# B&R Automation Studio project DeltaTestowa1 (part 2)

#### MainInitAction.st
```iecst
ACTION MainInitAction:

	MpPackMLCore_0.Enable := TRUE;
	MpPackMLMode_0.Enable := TRUE;
	MpDelta4Axis_0.Override := 100.0;
	MpDelta4Axis_0.Enable := TRUE;
	AxisParameters_0.Velocity := 50.0;
	AxisParameters_0.Acceleration := 20.0;
	AxisParameters_0.Deceleration := 20.0;

	AxisParameters_1.Velocity := 0.0;
	AxisParameters_1.Acceleration := 1.0;
	AxisParameters_1.Deceleration := 1.0;
	MpAxisBasic_0.Enable := TRUE;
	MpAxisBasic_1.Enable := TRUE;
	MpAxisBasic_Q1.Enable := TRUE;
	MpAxisBasic_Q2.Enable := TRUE;
	MpAxisBasic_Q3.Enable := TRUE;
	MpAxisBasic_Q4.Enable := TRUE;

	// dummy call of axis PVs just to avoid warning -2141192189 "The PV 'gAxisQx' does not exists" in logger
	gAxisQ1;
	gAxisQ2;
	gAxisQ3;
	gAxisQ4;

	IF DiagCpuIsARsim() THEN
		homingModeQ1.Homing.Mode := mcHOMING_DIRECT;
		homingModeQ2.Homing.Mode := mcHOMING_DIRECT;
		homingModeQ3.Homing.Mode := mcHOMING_DIRECT;
		homingModeQ4.Homing.Mode := mcHOMING_DIRECT;
	ELSE
		homingModeQ1.Homing.Mode := mcHOMING_DEFAULT;
		homingModeQ2.Homing.Mode := mcHOMING_DEFAULT;
		homingModeQ3.Homing.Mode := mcHOMING_DEFAULT;
		homingModeQ4.Homing.Mode := mcHOMING_DEFAULT;
	END_IF;

	//Activate block and set first state to Stopping (important, )
	MpPackMLMode_0.Activate := TRUE;
	MpPackMLMode_0.Stop := TRUE;

END_ACTION
```

#### MpPackCyclicAction.st
```iecst
ACTION MpPackCyclicAction:
	MpPackMLCore_0.MpLink := ADR(gPackMLCore);
	MpPackMLMode_0.MpLink := ADR(gPackMLCore);
	MpPackMLMode_0.ModeID := 1;

	MpPackMLMode_0.StateComplete := FALSE;
END_ACTION
```

#### AbortingAction.st
```iecst
ACTION AbortingAction:
	MpDelta4Axis_0.Power := FALSE;
	MpAxisBasic_0.Power := FALSE;
	ReadyMechanics := FALSE;
	AbortExecute := TRUE;
	CmdStart := FALSE;
	IF NOT MpDelta4Axis_0.PowerOn
		AND NOT MpAxisBasic_0.PowerOn THEN
		MpPackMLStateComplete(gPackMLCore,1);
	END_IF
END_ACTION
```

#### Action.st - not listed in the package file held
```iecst
ACTION ActionReseting:

	CASE RES_Step OF
		HOMING_DELTA:
			MpDelta4Axis_0.Home := TRUE;
			IF MpDelta4Axis_0.IsHomed THEN
				MpDelta4Axis_0.Home := FALSE;
				RES_Step := ACTIVATE_AXIS;
			END_IF

		ACTIVATE_AXIS:
			IF MpAxisBasic_0.Active AND MpDelta4Axis_0.Active THEN
				MpDelta4Axis_0.Power := TRUE;
				MpAxisBasic_0.Power := TRUE;
				MpAxisBasic_1.Power := TRUE; // axis not used, do not worry
				IF MpAxisBasic_0.PowerOn AND MpDelta4Axis_0.PowerOn THEN
					RES_Step := HOMING_AXIS;
				END_IF

			END_IF

		HOMING_AXIS:
			IF MpAxisBasic_0.PowerOn THEN
				MpAxisBasic_0.Home := TRUE;
				MpAxisBasic_1.Home := TRUE; // axis not used, do not worry
			END_IF;
			IF MpAxisBasic_0.IsHomed THEN
				MpAxisBasic_0.Home := FALSE;
				MpAxisBasic_1.Home := FALSE; // axis not used, do not worry
				RES_Step := COMPLETE_STATE;
			END_IF
		COMPLETE_STATE:
			MpPackMLStateComplete(gPackMLCore,1);

		END_CASE;
END_ACTION
```

### Program Logical/PickAndPlace/PrgPlace (IEC) - Place the products

#### Variables.var
```iecst
VAR
	P_Step : PlaceStepEnum;
	LastStep : PlaceStepEnum;
	Error : BOOL;
	PlaceHoldersSpacing : LREAL;
	LastPlaceHolderConveyorPosition : LREAL;
	ContainerID : UDINT;
	ElapsedDistance : LREAL;
END_VAR
(**)
(*Functionblocks*)
VAR
	MpPickRegister_0 : MpPickRegister;
	MpPickRegCreateContainer : MpPickRegCreateObject;
	MpPickRegGetObjectsContainer : MpPickRegGetObjects;
	MpPickRegDeleteTokens : MpPickRegDeleteObjects;
	Iterator : USINT;
	numberOfDeletes : USINT;
	TON_1 : TON;
	TON_0 : TON;
	OldTokenNumber : UDINT;
END_VAR
```

#### Main.st
```iecst
PROGRAM _INIT

    P_Step := P_WAIT_ENABLE;
    Error := FALSE;

	PlaceHoldersSpacing := 120; // distance between two consecutive place holders
	//numberOfDeletes := 2;
	gTokenNumber := 0;

END_PROGRAM

PROGRAM _CYCLIC

	IF NOT(gManualMode) THEN

	TON_0();
	TON_0.PT := T#5s;

    CASE P_Step OF
		P_WAIT_ENABLE:
			IF NOT AbortExecute AND NOT StopExecute AND NOT MpPickRegister_0.Error THEN
				P_Step := P_ENABLE_REGISTER_FB;
				StopExecutedPlace := FALSE;
				ClearingExecutedPlace := FALSE;
				MpPickRegister_0.ErrorReset := FALSE;
			END_IF

        P_ENABLE_REGISTER_FB:
            MpPickRegister_0.Enable := TRUE;
            P_Step := P_WAIT_ENABLE_REGISTER_FB;

        P_WAIT_ENABLE_REGISTER_FB:
            IF MpPickRegister_0.Active THEN
                P_Step := P_ENABLE_REGISTER_COMP;

            ELSIF MpPickRegister_0.Error THEN
                LastStep := P_Step;
                P_Step := P_ERROR;
            END_IF;

        P_ENABLE_REGISTER_COMP:
            MpPickRegister_0.RegisterEnable := TRUE;
            P_Step := P_WAIT_ENABLE_REGISTER_COMP;

        P_WAIT_ENABLE_REGISTER_COMP:
            IF MpPickRegister_0.RegisterActive THEN
                P_Step := P_ENABLE_ADD_REGISTER_FBS;

            ELSIF MpPickRegister_0.Error THEN
                LastStep := P_Step;
                P_Step := P_ERROR;
            END_IF;

        P_ENABLE_ADD_REGISTER_FBS:
            MpPickRegCreateContainer.Enable := TRUE;
			MpPickRegCreateContainer.Create := FALSE;
			MpPickRegGetObjectsContainer.Enable := TRUE;
			MpPickRegDeleteTokens.Enable := TRUE;
			P_Step := P_WAIT_ENABLE_ADD_REGISTER_FBS;

        P_WAIT_ENABLE_ADD_REGISTER_FBS:
            IF 	MpPickRegCreateContainer.Active THEN
                P_Step := P_WAIT_START_PROCESS;

            ELSIF MpPickRegCreateContainer.Error THEN
                LastStep := P_Step;
                P_Step := P_ERROR;
            END_IF;

        P_WAIT_START_PROCESS: // waits user start command and conveyor moving
            ReadyPlaceReg := TRUE;
            IF CmdStart AND ReadyToStart THEN
                P_Step := P_CREATE_OBJECTS;
            END_IF;

        (* We need to create positions (place holders) on place conveyor where to place picked objects *)
        P_CREATE_OBJECTS:

            ElapsedDistance := DistanceOverPeriod(PlaceConveyorPosition, LastPlaceHolderConveyorPosition, PlaceConveyorLength);

            IF (ElapsedDistance >= PlaceHoldersSpacing) THEN

                MpPickRegCreateContainer.Parameters.LatchedConveyor.Position := PlaceConveyorPosition;
                MpPickRegCreateContainer.Parameters.Mode := mpPICK_CREATE_CONTAINER_EMPTY;
				MpPickRegCreateContainer.Parameters.ObjectTypeName := 'MyContainer';
                MpPickRegCreateContainer.Parameters.Translation.X := 43;
				MpPickRegCreateContainer.Parameters.Translation.Y := 0;// in the middle of conveyor width
				MpPickRegCreateContainer.Parameters.Translation.Z := 2;
				ContainerID := MpPickRegCreateContainer.ObjectPositionId;
				MpPickRegCreateContainer.Create := TRUE;

				LastPlaceHolderConveyorPosition := MpPickRegCreateContainer.Parameters.LatchedConveyor.Position;
			ELSE
// Moze to trzeba rozwazyc ->ContainerID := MpPickRegCreateContainer.ObjectPositionId;
                MpPickRegCreateContainer.Create := FALSE;
            END_IF

        P_ERROR:
            Error := TRUE;
            ReadyPlaceReg := FALSE;

	END_CASE;

	IF StopExecute OR AbortExecute THEN
		ReadyPlaceReg := FALSE;
		P_Step := P_WAIT_ENABLE;
		StopExecutedPlace := TRUE;
	END_IF
	IF ClearingExecute THEN
		MpPickRegister_0.ErrorReset := TRUE;
		ClearingExecutedPlace := TRUE;
	END_IF

	MpPickRegGetObjectsContainer.Get := FALSE;
	MpPickRegDeleteTokens.Delete := FALSE;
	IF (MpPickRegGetObjectsContainer.Get = FALSE) THEN
		TON_0.IN := TRUE;

		IF TON_0.Q THEN
			MpPickRegGetObjectsContainer.Get := TRUE;
			TON_0.IN := FALSE;
		END_IF
	END_IF

	IF ContainerID > 0 THEN

		MpPickRegGetObjectsContainer.Parameters.DataAddress := ADR(gContainerInfo);
		MpPickRegGetObjectsContainer.Parameters.GetMode := mpPICK_GET_CONTAINER_CONTENT;
		MpPickRegGetObjectsContainer.Parameters.ObjectPositionId := ContainerID;
		MpPickRegGetObjectsContainer.Parameters.ObjectTypeName := 'MyContainer';
		MpPickRegGetObjectsContainer.Parameters.NumberOfObjectPositions := 4;
		MpPickRegGetObjectsContainer.MpLink := ADR(gPlaceRegister);
		MpPickRegGetObjectsContainer();

	END_IF;

		MpPickRegDeleteTokens.MpLink := ADR(gPlaceRegister);
		gTokenNumber := 0;

		FOR Iterator := 0 TO 3 DO
			IF (gContainerInfo[Iterator].ObjectPositionInfo = mpPICK_INFO_CONTAINED_OBJECT AND gDeleteObjects) THEN
				MpPickRegDeleteTokens.Parameters.ObjectTypeName := 'MyContainer';
				MpPickRegDeleteTokens.Parameters.ObjectPositionId := gContainerInfo[Iterator].ObjectPositionId;
				MpPickRegDeleteTokens.Delete := TRUE;
				numberOfDeletes := numberOfDeletes + 1;
			ELSE
				MpPickRegDeleteTokens.Parameters.ObjectTypeName := 'MyContainer';
				MpPickRegDeleteTokens.Parameters.ObjectPositionId := gContainerInfo[Iterator].ObjectPositionId;
				MpPickRegDeleteTokens.Delete := FALSE;
			END_IF;

			MpPickRegDeleteTokens();

			IF (gContainerInfo[Iterator].ObjectPositionInfo = mpPICK_INFO_CONTAINED_OBJECT) THEN
				gTokenNumber := gTokenNumber +1;
				IF OldTokenNumber <> gTokenNumber THEN
					gTokenOnConv := FALSE;
				END_IF

			END_IF

		END_FOR;
		IF numberOfDeletes > 0 THEN
			P_Step := P_WAIT_ENABLE;
			gTokenNumber := 0;
			numberOfDeletes := 0;
		END_IF
		gDeleteObjects := 0;
		OldTokenNumber := gTokenNumber;

		(* FB calls *)
		MpPickRegister_0.MpLink := ADR(gPlaceRegister);
		MpPickRegister_0();

		MpPickRegCreateContainer.MpLink := ADR(gPlaceRegister);
		MpPickRegCreateContainer();

	END_IF

END_PROGRAM
```

### Program Logical/PickAndPlace/PrgManual (IEC)

#### Types.typ
```iecst
TYPE
	MANUAL_ENUM :
		(
		HOMING := 1,
		XPOS := 2,
		XNEG := 3,
		YPOS := 4,
		YNEG := 5,
		ZPOS := 6,
		ZNEG := 7,
		OTHER := 8
		);
END_TYPE
```

#### Variables.var
```iecst
VAR
	HomeX : USINT;
	HomeY : USINT;
	HomingOffset : USINT;
	HomingVel : USINT;
	HomeZ : USINT;
	MoveXPos : BOOL;
	MoveXNeg : BOOL;
	MoveYPos : BOOL;
	MoveYNeg : BOOL;
	MoveZPos : BOOL;
	MoveZNeg : BOOL;
	XVel : USINT;
	YVel : USINT;
	ZVel : USINT;
	isMove : BOOL;
	ManualEnum : MANUAL_ENUM;
END_VAR
```

#### Main.st
```iecst
PROGRAM _INIT
	(* Insert code here *)
	gManualMode := 0;
	gMpDelta4AxisJog := FALSE;
	HomeX := 0;
	HomeY := 0;
	HomeZ := 120;
	HomingVel := 10;
	HomingOffset := 2;

END_PROGRAM

PROGRAM _CYCLIC
	IF gManualMode THEN
			//zapisac jako akcje:
		DeltaParamConnections.Jog.Velocity[0] := 0;
		DeltaParamConnections.Jog.Velocity[1] := 0;
		DeltaParamConnections.Jog.Velocity[2] := 0;

		IF isMove THEN
			gManualHoming := FALSE;
		END_IF;

		IF NOT isMove AND NOT gManualHoming THEN
			ManualEnum := 8;
		END_IF;

		IF gManualHoming THEN
			ManualEnum := 1;
		END_IF;

		gMpDelta4AxisEnable := TRUE;
		gMpDelta4AxisJog := TRUE;
		DeltaParamConnections.ManualMoveType := mcMOVE_RELATIVE;
		DeltaParamConnections.Jog.CoordSystem := mcTCS;
		DeltaParamConnections.CoordSystem := mcTCS;

		CASE ManualEnum OF
			HOMING:
				gMpDelta4AxisJog := TRUE;
				IF gTcpPositionX - HomeX > HomingOffset THEN
					DeltaParamConnections.Jog.Velocity[0] := -HomingVel;
				ELSIF HomeX - gTcpPositionX > HomingOffset THEN
					DeltaParamConnections.Jog.Velocity[0] := HomingVel;
				ELSIF gTcpPositionY - HomeY  > HomingOffset THEN
					DeltaParamConnections.Jog.Velocity[0] := 0;
					DeltaParamConnections.Jog.Velocity[1] := -HomingVel;
				ELSIF HomeY - gTcpPositionY > HomingOffset THEN
					DeltaParamConnections.Jog.Velocity[1] := HomingVel;
				ELSIF gTcpPositionZ - HomeZ > HomingOffset THEN
					DeltaParamConnections.Jog.Velocity[1] := 0;
					DeltaParamConnections.Jog.Velocity[2] := -HomingVel;
				ELSIF HomeZ - gTcpPositionZ > HomingOffset THEN
					DeltaParamConnections.Jog.Velocity[2] := HomingVel;
				ELSE
					DeltaParamConnections.Jog.Velocity[0] := 0;
					DeltaParamConnections.Jog.Velocity[1] := 0;
					DeltaParamConnections.Jog.Velocity[2] := 0;
				END_IF

			XPOS: DeltaParamConnections.Jog.Velocity[0] := XVel;
			XNEG: DeltaParamConnections.Jog.Velocity[0] := -XVel;
			YPOS: DeltaParamConnections.Jog.Velocity[1] := YVel;
			YNEG: DeltaParamConnections.Jog.Velocity[1] := -YVel;
			ZPOS: DeltaParamConnections.Jog.Velocity[2] := ZVel;
			ZNEG: DeltaParamConnections.Jog.Velocity[2] := -ZVel;
			OTHER: gMpDelta4AxisJog := FALSE;
			END_CASE

END_IF

END_PROGRAM
```

### Program Logical/PickAndPlace/Audyt (IEC)

#### Variables.var
```iecst
VAR
	MpAuditTrail_0 : MpAuditTrail;
	TypeVar : WSTRING[100];
	MessageVarStart : WSTRING[100];
	CommentVar : WSTRING[100];
	Zmienna : BOOL;
	DeleteAudit : BOOL;
	MpUserLogin_0 : MpUserLogin;
	R_TRIG_0 : R_TRIG;
	MessageVarLogin : WSTRING[100];
	MessageVarStop : WSTRING[100];
	MessageVarLogout : WSTRING[100];
	MessageVarCase : WSTRING[100];
	MessageVarAlarm : WSTRING[100];
	R_TRIG_1 : R_TRIG;
	R_TRIG_2 : R_TRIG;
	Login : BOOL;
	R_TRIG_3 : R_TRIG;
	Logout : BOOL;
	R_TRIG_4 : R_TRIG;
	R_TRIG_5 : R_TRIG;
	LoginFailed : BOOL;
	MessageVarLoginFailed : WSTRING[100];
	MessageVarManual : WSTRING[80];
	MessageVarAutomat : WSTRING[80];
	R_TRIG_6 : R_TRIG;
END_VAR
```

#### Main.st
```iecst
PROGRAM _INIT
	(* Insert code here *)
	MpAuditTrail_0.Enable := TRUE;
	Logout := FALSE;
END_PROGRAM

PROGRAM _CYCLIC
	//Wiadomości do audytu
	MessageVarStart := "Uruchomiono uklad";
	MessageVarStop := "Zatrzymano prace ukladu";
	MessageVarLogin := "Zalogowano uzytkownia";
	MessageVarLoginFailed := "Logowanie nie powiodlo sie";
	MessageVarLogout := "Wylogowano uzytkownika";
	MessageVarManual := "Zmiana trybu pracy na Manualny";
	MessageVarAutomat := "Zmiana trybu pracy na Automatyczny";
	//Wywoływanie audytu
	MpAuditTrail_0();
	MpAuditTrail_0.MpLink := ADR(gAuditTrail);
	MpAuditTrail_0.DeviceName := ADR('CF');
	//Usunięcie danych z audytu
	IF DeleteAudit THEN
		MpAuditClearBuffer(gAuditTrail);
		DeleteAudit := FALSE;
	END_IF;
	//Uruchomienie maszyny
	R_TRIG_0(CLK := CmdStart);
	IF R_TRIG_0.Q THEN
		MpAuditCustomEvent(gAuditTrail, TypeVar, MessageVarStart, CommentVar);
	END_IF;
	//Ausyt Stopu
	R_TRIG_1(CLK := StopExecute);
	IF R_TRIG_1.Q THEN
		MpAuditCustomEvent(gAuditTrail, TypeVar, MessageVarStop, CommentVar);
	END_IF;
	//Audyt zalogowania
	R_TRIG_2(CLK := Login);
	IF R_TRIG_2.Q THEN
		MpAuditCustomEvent(gAuditTrail, TypeVar, MessageVarLogin, CommentVar);
		Login := FALSE;
		Logout := FALSE;
	END_IF;
	//Audyt wylogowania
	R_TRIG_3(CLK := Logout);
	IF R_TRIG_3.Q THEN
		MpAuditCustomEvent(gAuditTrail, TypeVar, MessageVarLogout, CommentVar);
		Logout := FALSE;
	END_IF;
	//Audyt błąd logowania
	R_TRIG_4(CLK := LoginFailed);
	IF R_TRIG_4.Q THEN
		MpAuditCustomEvent(gAuditTrail, TypeVar, MessageVarLoginFailed, CommentVar);
		LoginFailed := FALSE;
	END_IF;
	//Audyt zmiany trybu pracy
	R_TRIG_5(CLK := gManualMode);
	IF R_TRIG_5.Q THEN
		MpAuditCustomEvent(gAuditTrail, TypeVar, MessageVarManual, CommentVar);
	END_IF;

	R_TRIG_6(CLK := NOT gManualMode);
	IF R_TRIG_6.Q THEN
		MpAuditCustomEvent(gAuditTrail, TypeVar, MessageVarAutomat, CommentVar);
	END_IF;

END_PROGRAM

PROGRAM _EXIT
	(* Insert code here *)

END_PROGRAM
```

### Program Logical/PickAndPlace/Alarmy (IEC)

#### Variables.var
```iecst
VAR
	MpAlarmXCore_0 : MpAlarmXCore;
	MpAlarmXHistory_0 : MpAlarmXHistory;
	ZmiennaTestowa : BOOL;
END_VAR
```

#### Main.st
```iecst
PROGRAM _INIT
	(* Insert code here *)
	MpAlarmXCore_0.Enable := TRUE;
	MpAlarmXCore_0.MpLink := ADR(gAlarmXCore);
	MpAlarmXCore_0();

	MpAlarmXHistory_0.Enable := TRUE;
	MpAlarmXHistory_0.MpLink := ADR(gAlarmXHistory);
	MpAlarmXHistory_0();
END_PROGRAM

PROGRAM _CYCLIC
	MpAlarmXCore_0.MpLink := ADR(gAlarmXCore);
	MpAlarmXHistory_0.MpLink := ADR(gAlarmXHistory);
	MpAlarmXHistory_0.DeviceName := ADR('CF');
	MpAlarmXCore_0();
	MpAlarmXHistory_0();

	IF ZmiennaTestowa THEN
		MpAlarmXSet(MpLink := gAlarmXCore, Name :='TestowyAlarm');
	END_IF;

	IF MpAlarmXHistory_0.Export THEN
		MpAlarmXHistory_0.Export := FALSE;
	END_IF;

END_PROGRAM

PROGRAM _EXIT
	(* Insert code here *)
	MpAlarmXCore_0.Enable := FALSE;
	MpAlarmXCore_0();
	MpAlarmXHistory_0.Enable := FALSE;
	MpAlarmXHistory_0();
END_PROGRAM
```

### Types.typ
```iecst
TYPE
	PML_CommandType : 	STRUCT  (*Commands structure*)
		UnitMode : DINT; (*Unit Mode target [Covered by MpPackMLCore PackTags]*)
		UnitModeChangeRequest : BOOL; (*Request Unit Mode change [Covered by MpPackMLCore PackTags]*)
		MachSpeed : REAL; (*Current machine speed [Primary packages/minute]*)
		MaterialInterlock : ARRAY[0..31]OF BOOL; (*Materials ready: MaterialInterlocks describes the status of the materials that are ready for processing*)
		CntrlCmd : DINT; (*Control Command [0=Undefined, 1=Reset, 2=Start, 3=Stop, 4=Hold, 5=Unhold, 6=Suspend, 7=Unsuspend, 8=Abort, 9=Clear] [Covered by MpPackMLCore PackTags]*)
		CmdChangeRequest : BOOL; (*State change request [Covered by MpPackMLCore PackTags]*)
		RemoteInterface : ARRAY[0..4]OF PML_RemoteInterfaceType; (*Upstream or downstream machine*)
		Parameter : ARRAY[0..4]OF PML_ParameterType; (*Parameter tags are associated to the end user supervisory interface*)
		Product : ARRAY[0..4]OF PML_ProductType; (*Product data type can be used for defining product and product processing parameter variables*)
	END_STRUCT;
	PML_StatusType : 	STRUCT  (*Status structure*)
		UnitModeCurrent : DINT; (*Unit Mode in current use [0=Invalid, 1=Production, 2=Maintenance, 3=Manual, 4-31=User definable) [Covered by MpPackMLCore PackTags]*)
		UnitModeRequested : BOOL; (*Requested Unit Mode change [Covered by MpPackMLCore PackTags]*)
		UnitModeChangeInProcess : BOOL; (*Requested Unit Mode change is in process [Covered by MpPackMLCore PackTags]*)
		StateCurrent : DINT; (*Current State Number [0=Undefined, 1=Clearing, 2=Stopped, 3=Starting, 4=Idle, 5=Suspended, 6=Execute, 7=Stopping, 8=Aborting, 9=Aborted, 10=Holding, 11=Held, 12=Unholding, 13=Suspending, 14=Unsuspending, 15=Resetting, 16=Completing, 17=Complete] [Covered by MpPackMLCore PackTags]*)
		StateRequested : DINT; (*Target State [0=Undefined, 1=Clearing, 2=Stopped, 3=Starting, 4=Idle, 5=Suspended, 6=Execute, 7=Stopping, 8=Aborting, 9=Aborted, 10=Holding, 11=Held, 12=Unholding, 13=Suspending, 14=Unsuspending, 15=Resetting, 16=Completing, 17=Complete]*)
		StateChangeInProcess : BOOL; (*State Change is in process [Covered by MpPackMLCore PackTags]*)
		MachSpeed : REAL; (*Current Machine Speed setpoint [Primary packages/minute]*)
		CurMachSpeed : REAL; (*Current Machine Speed real [Primary packages/minute]*)
		MaterialInterlock : ARRAY[0..31]OF BOOL; (*Materials ready: MaterialInterlocks describes the status of the materials that are ready for processing*)
		EquipmentInterlock : PML_EquipmentInterlockType; (*UpStream or downstream status*)
		RemoteInterface : ARRAY[0..4]OF PML_RemoteInterfaceType; (*Upstream or downstream machine*)
		Parameter : ARRAY[0..4]OF PML_ParameterType; (*Parameter tags are associated to the end user supervisory interface*)
		Product : ARRAY[0..4]OF PML_ProductType; (*Product data type can be used for displaying product and product processing parameter variables*)
	END_STRUCT;
	PML_AdminType : 	STRUCT  (*Administration structure*)
		Parameter : ARRAY[0..4]OF PML_ParameterType; (*Parameter tags associated to the local Interface are typically used for as parameters that are displayed or used on the unit locally, for example from an HMI*)
		Alarm : ARRAY[0..4]OF PML_AlarmType; (*Array of given size for machine fault number and messaging*)
		AlarmExtent : DINT; (*Extent of alarm array: the alarm extent is associated with the maximum number of alarms needed for the machine annunciation or reporting*)
		AlarmHistory : ARRAY[0..4]OF PML_AlarmType; (*Array of given size for machine fault number and messaging history*)
		AlarmHistoryExtent : DINT; (*Extent of alarm history array: the alarm history extent is associated with the maximum number of alarms needed to be archived or tagged as alarm history for the machine*)
		StopReason : PML_AlarmType; (*Machine stop reason is typically used for “First Out Fault” reporting and other stoppage events. The stop reason is the first event captured during an abort, held, suspended or stop event*)
		StopReasonExtent : DINT; (*Extent of stop reason array: the stop reason extent is associated with the maximum number of stop reasons needed to be archived or tagged as stop reasons for the machine*)
		Warning : PML_AlarmType; (*Machine warning are for general events that do not cause the machine to stop, but may require operator action as a stoppage may be imminent*)
		WarningExtent : DINT; (*The warning extent is associated with the maximum number of warnings needed to be archived or tagged as warnings for the machine*)
		ModeCurrentTime : ARRAY[0..31]OF DINT; (*Current amount of time (in sec) in any defined unit mode [Covered by MpPackMLCore PackTags]*)
		ModeCumulativeTime : ARRAY[0..31]OF DINT; (*Cumulative amount of time (in sec) in any defined unit mode [Covered by MpPackMLCore PackTags]*)
		StateCurrentTime : ARRAY[0..31]OF PML_ModeStateType; (*Current amount of time (in sec) in any defined state in any particular mode [Covered by MpPackMLCore PackTags]*)
		StateCumulativeTime : ARRAY[0..31]OF PML_ModeStateType; (*Cumulative amount of time (in sec) in any defined state in any particular mode since the last timer and counter reset was executed [Covered by MpPackMLCore PackTags]*)
		ProdConsumedCount : ARRAY[0..4]OF PML_ProdCountType; (*Material used / consumed in the production machine*)
		ProdProcessedCount : ARRAY[0..4]OF PML_ProdCountType; (*Number of products processed by the production machine*)
		ProdDefectiveCount : ARRAY[0..4]OF PML_ProdCountType; (*Product that is marked as defective in the production machine*)
		AccTimeSinceReset : DINT; (*Accumulative time since last reset [Covered by MpPackMLCore PackTags]*)
		MachDesignSpeed : REAL; (*Machine design speed [Primary Packages/minute]: maximum design speed of the machine in primary packages per minute for the package configuration being run*)
		StatesDisabled : DINT; (*States 1 to 17 of the PackML State Model can be disabled by turning on the corresponding bit in the INT.  Note that some state transition rules may over-ride the disable bits.  For Example, if HOLDING is not disabled, then HELD cannot be disabled*)
		PLCDateTime : PML_DateTimeType; (*Current Date and Time of the Programmable Logic Controller [Covered by MpPackMLCore PackTags]*)
	END_STRUCT;
	PML_RemoteInterfaceType : 	STRUCT  (*Upstream or downstream machine*)
		Number : DINT; (*Identification number of upstream or downstream unit machine*)
		ControlCmdNumber : DINT; (*Control command for upstream or downstream machine*)
		CmdValue : DINT; (*Control command value associated ControlCmdNumber*)
		Parameter : ARRAY[0..4]OF PML_ParameterType; (*Parameter tags associated to commanded remote interface*)
	END_STRUCT;
	PML_ParameterType : 	STRUCT  (*Parameter structure*)
		ID : DINT; (*ID value of Parameter*)
		Name : STRING[50]; (*String value assigned to Parameter*)
		Unit : STRING[5]; (*String value of Parameter units*)
		Value : REAL; (*Numeric value of Parameter*)
	END_STRUCT;
	PML_ProductType : 	STRUCT  (*Product structure*)
		ProductID : DINT; (*Structured array of Product ID#*)
		ProcessVariables : ARRAY[0..4]OF PML_ParameterType; (*Array of  data type Descriptor*)
		Ingredients : ARRAY[0..4]OF PML_IngredientsType; (*Structured Array for Ingredient Identification Parameters*)
	END_STRUCT;
	PML_AlarmType : 	STRUCT  (*Alarm structure*)
		Trigger : BOOL; (*Alarm Trigger should be turned on only when the alarm is currently active*)
		ID : DINT; (*Alarm message identification number *)
		Value : DINT; (*Alarm message number *)
		Message : STRING[80]; (*Alarm message*)
		Category : DINT; (*Alarm category: Category is used to identity what type of alarm has occurred (e.g. electrical, mechanical, materials, utilities, etc.)*)
		AlmDateTime : PML_DateTimeType; (*Structure of date and time in the alarm array to detail the date and time the alarm occurred*)
		AckDateTime : PML_DateTimeType; (*Structure of date and time in the alarm array to detail the date and time the alarm was acknowledged*)
	END_STRUCT;
	PML_IngredientsType : 	STRUCT  (*Ingredients structure*)
		IngredientID : DINT; (*The IngredientID is an arbitrary number associated with the raw material, or ingredient for a particular product number*)
		Parameter : ARRAY[0..4]OF PML_ParameterType; (*This array or structures is used for parameters associated with a particular ingredient or raw material used the processing of a particular product number*)
	END_STRUCT;
	PML_ProdCountType : 	STRUCT  (*Product count structure*)
		ID : DINT; (*This is the arbitrary (user defined) ID value of the consumed production material*)
		Name : STRING[80]; (*The name is used to literally describe the material ID, and its associated material*)
		Unit : STRING[5]; (*The unit tag is used to describe the names associated with a specific material used by the machine*)
		Count : DINT; (*The count value is used as a variable for displaying information about the amount of consumed production material*)
		AccCount : DINT; (*The accumulative count value is used as a variable for displaying information about the total amount of consumed production material*)
	END_STRUCT;
	PML_ModeStateType : 	STRUCT  (*Mode / State structure*)
		State : ARRAY[0..17]OF DINT; (*State inside each mode*)
	END_STRUCT;
	PML_EquipmentInterlockType : 	STRUCT  (*UpStream or downstream status*)
		Blocked : BOOL; (*This bit indicates that a downstream system is not able to accept product*)
		Starved : BOOL; (*This bit indicates that an upstream system is not able to supply product*)
	END_STRUCT;
	PML_DateTimeType : 	STRUCT  (*Date and time format*)
		Year : DINT; (*Date format: Year*)
		Month : DINT; (*Date format: Month*)
		Day : DINT; (*Date format: Day*)
		Hour : DINT; (*Time format: hours (24 hours format)*)
		Min : DINT; (*Time format: minutes*)
		Sec : DINT; (*Time format: seconds*)
		uSec : DINT; (*Time format: microseconds*)
	END_STRUCT;
END_TYPE
```

### Program Logical/PickAndPlace/PrgMechs

#### Variables.var
```iecst
VAR
	homingModeQ1 : MpAxisBasicParType;
	RC_Step : RCStepEnum;
	LastStep : RCStepEnum;
	DeltaParameters : MpDelta4AxisParType;
	MpAxisBasic_0 : MpAxisBasic;
	AxisParameters_0 : MpAxisBasicParType;
	MpAxisBasic_1 : MpAxisBasic;
	AxisParameters_1 : MpAxisBasicParType;
	MpAxisBasic_Q1 : MpAxisBasic;
	MpAxisBasic_Q2 : MpAxisBasic;
	MpAxisBasic_Q3 : MpAxisBasic;
	Delta : MpAxisBasic;
	MpAxisBasic_Q4 : MpAxisBasic;
	homingModeQ3 : MpAxisBasicParType;
	homingModeQ4 : MpAxisBasicParType;
	homingModeQ2 : MpAxisBasicParType;
	MpDelta4Axis_0 : MpDelta4Axis;
END_VAR
```

#### Main.st
```iecst
PROGRAM _INIT

    MpDelta4Axis_0.Override := 100.0;
    MpDelta4Axis_0.Enable   := TRUE;

    AxisParameters_0.Velocity     := 50.0;
    AxisParameters_0.Acceleration := 20.0;
    AxisParameters_0.Deceleration := 20.0;

    AxisParameters_1.Velocity     := 0.0;
    AxisParameters_1.Acceleration := 1.0;
    AxisParameters_1.Deceleration := 1.0;

    MpAxisBasic_0.Enable := TRUE;
    MpAxisBasic_1.Enable := TRUE;

    // dummy call of axis PVs just to avoid warning -2141192189 "The PV 'gAxisQx' does not exists" in logger
    gAxisQ1;
    gAxisQ2;
    gAxisQ3;
	gAxisQ4;

END_PROGRAM

PROGRAM _CYCLIC

    (* Prepare mechanics: Robot & conveyors *)
    CASE RC_Step OF

        (* first preparing robot *)
        RC_WAIT_ENABLE:
            IF MpDelta4Axis_0.Active THEN
                RC_Step := RC_POWER_ROBOT;
            END_IF

        RC_POWER_ROBOT:
            MpDelta4Axis_0.Power := TRUE;
            IF MpDelta4Axis_0.PowerOn THEN
                RC_Step := RC_HOME_ROBOT;
            END_IF

        RC_HOME_ROBOT:
			MpDelta4Axis_0.Home := TRUE;
			IF MpDelta4Axis_0.IsHomed THEN
				MpDelta4Axis_0.Home := FALSE;
                RC_Step := RC_ROBOT_READY;
           END_IF

        RC_ROBOT_READY:
            RC_Step := RC_WAIT_ENABLE_AXIS_FB;

        (* preparing conveyors *)
        RC_WAIT_ENABLE_AXIS_FB:
            IF MpAxisBasic_0.Active THEN
                IF MpAxisBasic_1.Active THEN
                    RC_Step := RC_POWER_AXIS;
                END_IF
            ELSIF MpAxisBasic_0.Error OR MpAxisBasic_1.Error THEN
                LastStep := RC_Step;
                RC_Step  := RC_ERROR;
            END_IF;

        RC_POWER_AXIS:
            MpAxisBasic_0.Power := TRUE;
            MpAxisBasic_1.Power := TRUE;
            RC_Step := RC_WAIT_POWER_AXIS;

        RC_WAIT_POWER_AXIS:
            IF MpAxisBasic_0.PowerOn THEN
                IF MpAxisBasic_1.PowerOn THEN
                    RC_Step := RC_HOME_AXIS;
                END_IF
            ELSIF MpAxisBasic_0.Error OR MpAxisBasic_1.Error THEN
                LastStep := RC_Step;
                RC_Step  := RC_ERROR;
            END_IF;

        RC_HOME_AXIS:
            MpAxisBasic_0.Home := TRUE;
            MpAxisBasic_1.Home := TRUE;
            RC_Step := RC_WAIT_HOME_AXIS;

        RC_WAIT_HOME_AXIS:
			IF MpAxisBasic_0.IsHomed THEN
				IF MpAxisBasic_0.IsHomed THEN
                    MpAxisBasic_0.Home := FALSE;
                    MpAxisBasic_1.Home := FALSE;
					RC_Step := RC_READY;

                END_IF
			ELSIF MpAxisBasic_0.Error OR MpAxisBasic_1.Error THEN
				LastStep := RC_Step;
				RC_Step  := RC_ERROR;
			END_IF;

        RC_READY:
            ReadyMechanics := TRUE;
            IF CmdStart AND ReadyToStart THEN
                RC_Step := RC_START_PROCESS;
            END_IF;

        (* start conveyors to move *)
        RC_START_PROCESS:
            MpAxisBasic_0.MoveVelocity := TRUE;
            MpAxisBasic_1.MoveVelocity := TRUE;
            RC_Step := RC_WAIT_PROCESS_STARTED;

        RC_WAIT_PROCESS_STARTED:
            IF MpAxisBasic_0.Info.PLCopenState = mcAXIS_CONTINUOUS_MOTION THEN
                IF MpAxisBasic_1.Info.PLCopenState = mcAXIS_CONTINUOUS_MOTION THEN
                    RC_Step := RC_PROCESSING;
                END_IF
            ELSIF MpAxisBasic_0.Error OR MpAxisBasic_1.Error THEN
                LastStep := RC_Step;
                RC_Step  := RC_ERROR;
            END_IF;

        RC_PROCESSING:
            IF MpAxisBasic_0.Error OR MpAxisBasic_1.Error THEN
                LastStep := RC_Step;
                RC_Step  := RC_ERROR;
            END_IF;

        RC_ERROR:
            ReadyMechanics := FALSE;

    END_CASE

    ReadyToStart := ReadyMechanics AND ReadyPickReg AND ReadyPlaceReg AND ReadyPickCore;

    (* Call FBs *)
    MpDelta4Axis_0.MpLink     := ADR(g4AxDeltaA);
    MpDelta4Axis_0.Parameters := ADR(DeltaParameters);
    MpDelta4Axis_0();

    MpAxisBasic_0.MpLink     := ADR(gAxis_1);
    MpAxisBasic_0.Parameters := ADR(AxisParameters_0);
    MpAxisBasic_0();

    MpAxisBasic_1.MpLink     := ADR(gAxis_2);
    MpAxisBasic_1.Parameters := ADR(AxisParameters_1);
    MpAxisBasic_1();

    PickConveyorPosition  := MpAxisBasic_0.Position;
    PlaceConveyorPosition := MpAxisBasic_1.Position;

END_PROGRAM
```

### Program Logical/PickAndPlace/UsersMenagment

#### Main.st
```iecst
PROGRAM _INIT
	(* Insert code here *)
	MpAlarmXCore_0.Enable := TRUE;
	MpAlarmXCore_0.MpLink := ADR(gAlarmXCore);
	MpAlarmXCore_0();

	MpAlarmXHistory_0.Enable := TRUE;
	MpAlarmXHistory_0.MpLink := ADR(gAlarmXCore);
	MpAlarmXHistory_0();
END_PROGRAM

PROGRAM _CYCLIC
	MpAlarmXCore_0.MpLink := ADR(gAlarmXCore);
	MpAlarmXHistory_0.MpLink := ADR(gAlarmXHistory);

	MpAlarmXCore_0();
	MpAlarmXHistory_0();

	IF ZmiennaTestowa THEN
		MpAlarmXSet(MpLink := gAlarmXCore, Name :='TestowyAlarm');
	END_IF;

END_PROGRAM

PROGRAM _EXIT
	(* Insert code here *)
	MpAlarmXCore_0.Enable := FALSE;
	MpAlarmXCore_0();
	MpAlarmXHistory_0.Enable := FALSE;
	MpAlarmXHistory_0();
END_PROGRAM
```

- Visualisation Logical/mappView (not shown)

- Project.language (not shown)

### Program Logical/Camera/Vision (IEC)

#### Main.st - Init, cyclic, exit code
```iecst
PROGRAM _INIT
	(* Insert code here *)

		//Config camera triggered by position of axis
	AcquisitionParameters.StartPosition :=0;
	AcquisitionParameters.Period := 160;
	AcquisitionParameters.AcquisitionPositions[0] := 80;

	//advanced settings
	AdvancedParameters.DisableNegativeDirection := FALSE;
	AdvancedParameters.AddOutputCompensation :=0.5;
	AdvancedParameters.AddPositionCompensation:=0.5;

	ViAxisAcquisition_0.Update:=0;
	ViAxisAcquisition_0.MpLink:=ADR(gCamera);

	ViAxisAcquisition_0.AcquisitionParameters:= AcquisitionParameters;
	ViAxisAcquisition_0.AdvancedParameters := AdvancedParameters;
	MakingPhoto := ViAxisAcquisition_0.InOperation;

	//Config img Acquisition
	ImageGetter.MpLink:= ADR(gCamera);
	ImageGetter.Buffer:=ADR(BufferForBinaryImageData);
	ImageGetter.BufferSize:= SIZEOF(BufferForBinaryImageData);
	ImageGetter.Type:= viBASE_IMAGE_TYPE_JPG;
	ImageGetter.QualityLevel:=10;

	//AdvancedParameters.

	Cam.Parameters.MinScore := 80;

END_PROGRAM

PROGRAM _CYCLIC
	(* Insert code here *)

	//Main acquisition
	gMakeToken:=0;
	IF Cam.Status.IsCameraReady AND gIsConvHomed THEN
		ViAxisAcquisition_0.Enable := TRUE;
		// Token pos
		IF EDGENEG(gIsCameraActive) THEN
		IF Cam.Camera_Output.NumResults > 0 THEN

			RotationPeriod :=360/ConvVelocityDegrees;
			gToken_X := 120 - (((Cam.Camera_Output.PosMatchX*313)/1.7/108000)-100);
			gToken_Y := 165 - (((Cam.Camera_Output.PosMatchY*174)/195200)*1.83) + 45+ ((UINT_TO_REAL(Cam.Camera_Output.ProcesingTime)/1000.0)*ConvVelocityDegrees) ;
			gMakeToken:=1;

			END_IF

			ImageGetter.Execute:=TRUE;

		END_IF

	END_IF

	// Measurements conversion

	// Token operations (sim creation; pos updater)

	//GetImage
	IF EDGEPOS(ImageGetter.Done) THEN
		strcpy(ADR(CameraImageURL),ADR('<image x=$'0$' y=$'0$' width=$'615px$' height=$'630px$' href=$'data:image/jpeg;base64,')); // Start of the image element with image dimensions as set in the vision application.
		ImgTransfer.pDest :=ADR(BufferForBase64EncodedImageData);
		Buffersize := SIZEOF(BufferForBase64EncodedImageData);
		Bufferlen := strlen(ADR(BufferForBase64EncodedImageData));
		Stringlen := strlen(ADR('$' />'));
		ImgTransfer.destSize := Buffersize - Bufferlen - Stringlen;
		ImgTransfer.pSrc := ADR(BufferForBinaryImageData);
		ImgTransfer.srcLen := ImageGetter.BufferLen;
		ImgTransfer.enable := TRUE;
		ImgTransfer();

		strcat(ADR(CameraImageURL),ADR(BufferForBase64EncodedImageData));
		strcat(ADR(CameraImageURL),ADR('$' />')) ; // Completion of the image element

	END_IF

	IF ImageGetter.Done THEN
		ImageGetter.Execute := FALSE;
		END_IF

	ViAxisAcquisition_0();
	ImageGetter();

END_PROGRAM

PROGRAM _EXIT
	(* Insert code here *)

END_PROGRAM
```

#### Variables.var - Local variables
```iecst
VAR
	OldPhotosNum : USINT;
	Cam : Camera;
	ViAxisAcquisition_0 : ViBaseAxisBasedAcquisition;
	AcquisitionParameters : ViBaseAxBsdAcqAcqParType;
	AdvancedParameters : ViBaseAxBsdAcqAdvParType;
	MakingPhoto : BOOL;
	CameraStatus : UDINT;
	RotationPeriod : REAL;
	ImageGetter : ViBaseGetImage;
	BufferForBinaryImageData : ARRAY[0..2500000] OF USINT;
	BufferForBase64EncodedImageData : STRING[2500000];
	ImgTransfer : httpEncodeBase64;
	Buffersize : UDINT;
	Bufferlen : UDINT;
	Stringlen : UDINT;
	CameraImageURL : STRING[2500000];
END_VAR
```

#### Camera.typ
```iecst
TYPE
	Camera : 	STRUCT
		Cmd : Cmd;
		Parameters : Parameters;
		Status : Status;
		Camera_Output : Camera_Output;
	END_STRUCT;
	Parameters : 	STRUCT
		SetFocus : UINT := 45000;
		ExposureTime : UDINT := 10000;
		FlashColor : USINT := 99;
		FlashSegment : USINT := 15;
		MinScore : USINT;
	END_STRUCT;
	Cmd : 	STRUCT
		Trigger : BOOL;
		Enable_Matching : BOOL := 1;
	END_STRUCT;
	Status : 	STRUCT
		AquisitionComplete : BOOL;
		IsCameraReady : BOOL;
	END_STRUCT;
	Camera_Output : 	STRUCT
		PosMatchX : DINT;
		PosMatchY : DINT;
		NumResults : USINT;
		PhotosNum : USINT;
		ProcesingTime : UINT;
	END_STRUCT;
END_TYPE
```

### Program Logical/Camera/Kamera (IEC)

#### Main.ab - Init, cyclic, exit code
```automation-basic
PROGRAM _INIT
	(* Insert code here *)

	ViAxisAcquisition_0.MpLink:=ADR(gCamera);
	ViAxisAcquisition_0.Enable := TRUE;
	ViAxisAcquisition_0.AcquisitionParameters:= AcquisitionParameters;
	ViAxisAcquisition_0.AdvancedParameters := AdvancedParameters;
	MakingPhoto := ViAxisAcquisition_0.InOperation

	//Config camera triggered by position of axis
	AcquisitionParameters.StartPosition :=0;
	AcquisitionParameters.Period := 160;
	AcquisitionParameters.AcquisitionPositions[0] := 80;
	//AdvancedParameters.

END_PROGRAM

PROGRAM _CYCLIC
	(* Insert code here *)

END_PROGRAM

PROGRAM _EXIT
	(* Insert code here *)

END_PROGRAM
```

#### Variables.var - Local variables
```iecst
VAR
	MpLink : ViComponentType;
	Enable : BOOL;
	AcquisitionParameters : ViBaseAxBsdAcqAcqParType;
	AdvancedParameters : ViBaseAxBsdAcqAdvParType;
	ViAxisAcquisition_0 : ViBaseAxisBasedAcquisition;
	MakingPhoto : BOOL;
END_VAR
```

### McAcpTrakCfg.typ
```iecst
TYPE
	McASMTrkSegType : STRUCT (*Segments which define the track*)
		SegmentReference : McCfgUnboundedArrayType; (*Name of the referenced segment component*)
	END_STRUCT;
	McASMTrkPosEnum :
		( (*Position selector setting*)
		mcASMTP_ABS := 0, (*Absolute - Absolute position in the workspace*)
		mcASMTP_REL_TO_ONE_SEG := 1, (*Relative to one segment - Position relative to one segment*)
		mcASMTP_REL_TO_TWO_SEG := 2 (*Relative to two segments - Position relative to two segments*)
		);
	McASMTrkPosAbsSegCntDirEnum :
		( (*Count direction of the track in the workspace*)
		mcASMTPASCD_RIGHT_TO_LFT := 0, (*Right to left - Positive count direction is from the right to the left side*)
		mcASMTPASCD_LFT_TO_RIGHT := 1 (*Left to right - Positive count direction is from the left to the right side*)
		);
	McASMSegPosRelToEnum :
		( (*Absolute position from which the position is counted*)
		mcASMSPRT_ST_OF_SEG := 0, (*Start of segment - Positive from start of segment*)
		mcASMSPRT_END_OF_SEG := 1 (*End of segment - Negative from end of segment*)
		);
	McASMTrkPosAbsType : STRUCT (*Type mcASMTP_ABS settings*)
		SegmentReference : STRING[250]; (*Name of the referenced segment component*)
		SegmentCountDirection : McASMTrkPosAbsSegCntDirEnum; (*Count direction of the track in the workspace*)
		Position : LREAL; (*Position on the segment [Measurement units]*)
		PositionRelativeTo : McASMSegPosRelToEnum; (*Absolute position from which the position is counted*)
		Translation : McCfgTransXYZType; (*Translation parameters*)
		Orientation : McCfgOrientType; (*Orientation parameters*)
	END_STRUCT;
	McASMSegType : STRUCT (*Segment of the new track*)
		SegmentReference : STRING[250]; (*Name of the referenced segment component*)
		Position : LREAL; (*Position on the segment [Measurement units]*)
		PositionRelativeTo : McASMSegPosRelToEnum; (*Absolute position from which the position is counted*)
	END_STRUCT;
	McASMTrkPosRelOneType : STRUCT (*Type mcASMTP_REL_TO_ONE_SEG settings*)
		SegmentTrack : McASMSegType; (*Segment of the new track*)
		SegmentExistingTrack : McASMSegType; (*The new track is relative to this segment*)
	END_STRUCT;
	McASMTrkPosRelTwoAlignType : STRUCT (*Alignment of the new track to the first segment*)
		SegmentRefTrack : STRING[250]; (*Name of the referenced segment component*)
		SegmentRefExistingTrack : STRING[250]; (*Name of the referenced segment component*)
	END_STRUCT;
	McASMTrkPosRelTwoType : STRUCT (*Type mcASMTP_REL_TO_TWO_SEG settings*)
		AlignmentFirst : McASMTrkPosRelTwoAlignType; (*Alignment of the new track to the first segment*)
		AlignmentSecond : McASMTrkPosRelTwoAlignType; (*Alignment of the new track to the second segment*)
	END_STRUCT;
	McASMTrkPosType : STRUCT (*Position of the track in the workspace*)
		Type : McASMTrkPosEnum; (*Position selector setting*)
		Absolute : McASMTrkPosAbsType; (*Type mcASMTP_ABS settings*)
		RelativeToOneSegment : McASMTrkPosRelOneType; (*Type mcASMTP_REL_TO_ONE_SEG settings*)
		RelativeToTwoSegments : McASMTrkPosRelTwoType; (*Type mcASMTP_REL_TO_TWO_SEG settings*)
	END_STRUCT;
	McASMTrkType : STRUCT (*Track definition*)
		Segments : McASMTrkSegType; (*Segments which define the track*)
		Position : McASMTrkPosType; (*Position of the track in the workspace*)
	END_STRUCT;
	McASMTrksType : STRUCT (*Settings for all tracks that define the assembly*)
		TrackSeparation : LREAL; (*Gap between the stator surfaces of opposite tracks [Measurement units]*)
		Track : McCfgUnboundedArrayType; (*Track definition*)
	END_STRUCT;
	McASMCSSActSegSimOnPLCEnum :
		( (*All segments of the assembly are simulated on the PLC*)
		mcASMCSSASSOP_OFF := 0, (*Off - The segments are not simulated on the PLC*)
		mcASMCSSASSOP_ON := 1 (*On - The segments are simulated on the PLC*)
		);
	McASMCSSCogSegTransCompEnum :
		( (*Cogging at segment transition compensation selector setting*)
		mcASMCSSCSTC_INACT := 0, (*Inactive - No compensation of cogging at segment transition*)
		mcASMCSSCSTC_ACT := 1 (*Active - Compensation of cogging at segment transition*)
		);
	McASMCSSCogSegTransCompActType : STRUCT (*Type mcASMCSSCSTC_ACT settings*)
		UpperVelocityLimit : REAL; (*Beneath this limit the cogging compensation at segment transition will be applied. [m/s]*)
	END_STRUCT;
	McASMCSSCogSegTransCompType : STRUCT (*Compensation of cogging at segment transition to reduce lag and speed error*)
		Type : McASMCSSCogSegTransCompEnum; (*Cogging at segment transition compensation selector setting*)
		Active : McASMCSSCogSegTransCompActType; (*Type mcASMCSSCSTC_ACT settings*)
	END_STRUCT;
	McASMCSSElongationCompEnum :
		( (*Compensation of segment elongation due to change of temperature*)
		mcASMCSSEC_INACT := 0, (*Inactive - No compensation of segment elongation*)
		mcASMCSSEC_ACT := 1 (*Active - Compensation of segment elongation*)
		);
	McASMCSSStopReacEnum :
		( (*Stop reaction selector setting*)
		mcASMCSSSR_INDUCT_HALT := 0, (*Induction halt - Shuttle stop by setting current in all segment coils*)
		mcASMCSSSR_COAST_TO_STANDSTILL := 1 (*Coast to standstill - Shuttle stop by reseting current in all segment coils - stop by friction*)
		);
	McASMCSSStopReacType : STRUCT (*Reaction in case of certain stop conditions*)
		Type : McASMCSSStopReacEnum; (*Stop reaction selector setting*)
	END_STRUCT;
	McASMCSSSpdFltrEnum :
		( (*Speed filter selector setting*)
		mcASMCSSSF_NOT_USE := 0, (*Not used - Speed filter disabled*)
		mcASMCSSSF_LP_1ST_ORD := 1 (*Lowpass 1st order - Lowpass 1st order speed filter*)
		);
	McASMCSSSpdFltrLP1stOrdType : STRUCT (*Type mcASMCSSSF_LP_1ST_ORD settings*)
		FilterTime : REAL; (*Filter time constant [s]*)
	END_STRUCT;
	McASMCSSSpdFltrType : STRUCT (*Filter for actual speed calculation*)
		Type : McASMCSSSpdFltrEnum; (*Speed filter selector setting*)
		Lowpass1stOrder : McASMCSSSpdFltrLP1stOrdType; (*Type mcASMCSSSF_LP_1ST_ORD settings*)
	END_STRUCT;
	McASMCSSCtrlSetPosType : STRUCT (*Position controller parameters*)
		ProportionalGain : REAL; (*Proportional amplification [1/s]*)
	END_STRUCT;
	McASMCSSCtrlSetSpdType : STRUCT (*Speed controller parameters*)
		ProportionalGain : REAL; (*Proportional amplification [N s/m]*)
		IntegrationTime : REAL; (*Integral action time [s]*)
	END_STRUCT;
	McASMCSSCtrlSetFFwdType : STRUCT (*Force feed forward controller parameters*)
		TotalMass : REAL; (*Total mass [kg]*)
		ForcePositive : REAL; (*Force in positive direction [N]*)
		ForceNegative : REAL; (*Force in negative direction [N]*)
		SpeedForceFactor : REAL; (*Speed force factor [N s/m]*)
		ForceLoad : REAL; (*External load [N]*)
	END_STRUCT;
	McASMCSSCtrlSetType : STRUCT (*Axis controller parameters*)
		Position : McASMCSSCtrlSetPosType; (*Position controller parameters*)
		Speed : McASMCSSCtrlSetSpdType; (*Speed controller parameters*)
		FeedForward : McASMCSSCtrlSetFFwdType; (*Force feed forward controller parameters*)
	END_STRUCT;
	McASMCSSMoveErrLimType : STRUCT (*Limit values which lead to a stop reaction in case they are exceeded*)
		PositionError : LREAL; (*Lag error limit for stop of a movement [Measurement units]*)
		VelocityError : LREAL; (*Velocity lag error limit for stop of a movement [Measurement units/s]*)
	END_STRUCT;
	McASMCSSDivForceType : STRUCT (*Diverter parameters*)
		ForceOverrideFactor : REAL; (*Override the default diverter force set value*)
	END_STRUCT;
	McASMCSSCPDPSType : STRUCT (*Parameter set 0*)
		Controller : McASMCSSCtrlSetType; (*Axis controller parameters*)
		MovementErrorLimits : McASMCSSMoveErrLimType; (*Limit values which lead to a stop reaction in case they are exceeded*)
		Diverter : McASMCSSDivForceType; (*Diverter parameters*)
	END_STRUCT;
	McASMCSSCPAPSEnum :
		( (*Additional parameter sets selector setting*)
		mcASMCSSCPAPS_NOT_USE := 0, (*Not used - Additional parameter sets are not used*)
		mcASMCSSCPAPS_USE := 1 (*Used - Additional parameter sets are used*)
		);
	McASMCSSCPAPSUseParSetCtrlEnum :
		( (*Controller selector setting*)
		mcASMCSSCPAPSUPSC_USE_DEF_VAL := 0, (*Use default values - Use the values from the default parameter set*)
		mcASMCSSCPAPSUPSC_USE_EXP_VAL := 1 (*Use explicit values - Define values for this parameter set*)
		);
	McASMCSSCPAPSUseParSetCtrlType : STRUCT (*Axis controller parameters*)
		Type : McASMCSSCPAPSUseParSetCtrlEnum; (*Controller selector setting*)
		UseExplicitValues : McASMCSSCtrlSetType; (*Type mcASMCSSCPAPSUPSC_USE_EXP_VAL settings*)
	END_STRUCT;
	McASMCSSCPAPSUPSMoveErrLimEnum :
		( (*Movement error limits selector setting*)
		mcASMCSSCPAPSUPSMEL_USE_DEF_VAL := 0, (*Use default values - Use the values from the default parameter set*)
		mcASMCSSCPAPSUPSMEL_USE_EXP_VAL := 1 (*Use explicit values - Define values for this parameter set*)
		);
	McASMCSSCPAPSUPSMoveErrLimType : STRUCT (*Limit values which lead to a stop reaction in case they are exceeded*)
		Type : McASMCSSCPAPSUPSMoveErrLimEnum; (*Movement error limits selector setting*)
		UseExplicitValues : McASMCSSMoveErrLimType; (*Type mcASMCSSCPAPSUPSMEL_USE_EXP_VAL settings*)
	END_STRUCT;
	McASMCSSCPAPSUPSDivEnum :
		( (*Diverter selector setting*)
		mcASMCSSCPAPSUPSDIV_USE_DEF_VAL := 0, (*Use default values - Use the values from the default parameter set*)
		mcASMCSSCPAPSUPSDIV_USE_EXP_VAL := 1 (*Use explicit values - Define values for this parameter set*)
		);
	McASMCSSCPAPSUPSDivType : STRUCT (*Diverter parameters*)
		Type : McASMCSSCPAPSUPSDivEnum; (*Diverter selector setting*)
		UseExplicitValues : McASMCSSDivForceType; (*Type mcASMCSSCPAPSUPSDIV_USE_EXP_VAL settings*)
	END_STRUCT;
	McASMCSSCPAPSUseParSetType : STRUCT (*Additional parameter set*)
		Controller : McASMCSSCPAPSUseParSetCtrlType; (*Axis controller parameters*)
		MovementErrorLimits : McASMCSSCPAPSUPSMoveErrLimType; (*Limit values which lead to a stop reaction in case they are exceeded*)
		Diverter : McASMCSSCPAPSUPSDivType; (*Diverter parameters*)
	END_STRUCT;
	McASMCSSCPAPSUseType : STRUCT (*Type mcASMCSSCPAPS_USE settings*)
		ParameterSet : McCfgUnboundedArrayType; (*Additional parameter set*)
	END_STRUCT;
	McASMCSSCPAPSType : STRUCT (*Enable additional parameter sets that can be switched during runtime*)
		Type : McASMCSSCPAPSEnum; (*Additional parameter sets selector setting*)
		Used : McASMCSSCPAPSUseType; (*Type mcASMCSSCPAPS_USE settings*)
	END_STRUCT;
	McASMCSSCtrlParType : STRUCT (*Segment controller parameters*)
		DefaultParameterSet : McASMCSSCPDPSType; (*Parameter set 0*)
		AdditionalParameterSets : McASMCSSCPAPSType; (*Enable additional parameter sets that can be switched during runtime*)
	END_STRUCT;
	McASMCSSScpErrReacEnum :
		( (*Setting for the minimal error reaction scope with segment errors*)
		mcASMCSSSER_ASM := 0, (*Assembly - Error reaction triggered for the whole assembly*)
		mcASMCSSSER_SEG := 1 (*Segment - Error reaction triggered for the faulty segment, if type of error permits that*)
		);
	McASMCSSPosCtrlLagMonEnum :
		( (*Position controller lag monitor selector setting*)
		mcASMCSSPCLM_INACT := 0, (*Inactive - The position controller lag is not cyclically monitored*)
		mcASMCSSPCLM_ACT := 1 (*Active - The position controller lag is cyclically monitored*)
		);
	McASMCSSPosCtrlLagMonActType : STRUCT (*Type mcASMCSSPCLM_ACT settings*)
		WarningLimit : REAL; (*Limit value which leads to a position controller lag warning in case it is exceeded [m]*)
	END_STRUCT;
	McASMCSSPosCtrlLagMonType : STRUCT (*Setting for the position controller lag monitor*)
		Type : McASMCSSPosCtrlLagMonEnum; (*Position controller lag monitor selector setting*)
		Active : McASMCSSPosCtrlLagMonActType; (*Type mcASMCSSPCLM_ACT settings*)
	END_STRUCT;
	McASMCSSDiverterType : STRUCT (*Diverter parameters*)
		WeakeningEndOverrideFactor : REAL; (*Override the default endpoint where the magnetic field is weakened to actively force a shuttle to the desired track side*)
		StrengtheningEndOverrideFactor : REAL; (*Override the default endpoint where the magnetic field is strengthened to actively force a shuttle to the desired track side*)
	END_STRUCT;
	McASMCSSType : STRUCT (*Common settings for all segments in the assembly*)
		ActivateSegmentSimulationOnPLC : McASMCSSActSegSimOnPLCEnum; (*All segments of the assembly are simulated on the PLC*)
		CoggingSegTransCompensation : McASMCSSCogSegTransCompType; (*Compensation of cogging at segment transition to reduce lag and speed error*)
		ElongationCompensation : McASMCSSElongationCompEnum; (*Compensation of segment elongation due to change of temperature*)
		StopReaction : McASMCSSStopReacType; (*Reaction in case of certain stop conditions*)
		SpeedFilter : McASMCSSSpdFltrType; (*Filter for actual speed calculation*)
		ControllerParameters : McASMCSSCtrlParType; (*Segment controller parameters*)
		ScopeErrorReaction : McASMCSSScpErrReacEnum; (*Setting for the minimal error reaction scope with segment errors*)
		ShuttleIdentificationTime : UINT; (*Time period in which the identification of the shuttles must take place during power-on [s]*)
		PositionControllerLagMonitor : McASMCSSPosCtrlLagMonType; (*Setting for the position controller lag monitor*)
		Diverter : McASMCSSDiverterType; (*Diverter parameters*)
	END_STRUCT;
	McASMShConFunEnum :
		( (*Activate for usage of shuttle convoys*)
		mcASMSCF_INACT := 0, (*Inactive - Convoy functionality is not used*)
		mcASMSCF_ACT := 1 (*Active - Convoy functionality is used*)
		);
	McASMShSSASEnum :
		( (*Switch sector after stop selector setting*)
		mcASMSSSAS_SW_ONTO_SEG_SEC := 0, (*Switch onto segment sector - Switch onto the segment sector*)
		mcASMSSSAS_AUT_ATT := 1, (*Auto attach - Autoattach*)
		mcASMSSSAS_RMN_ON_INT_SEC := 2 (*Remain on internal sector - Remain on the internal sector*)
		);
	McASMShSSASSwOntoSegSecScpEnum :
		( (*The scope of the setting*)
		mcASMSSSASSOSSS_SH_ONLY := 0, (*Shuttle only - Switch the shuttle or the trivial convoy onto the segment sector*)
		mcASMSSSASSOSSS_ALL := 1 (*All - Switch the shuttle or convoy onto the segment sector*)
		);
	McASMShSSASSwOntoSegSecType : STRUCT (*Type mcASMSSSAS_SW_ONTO_SEG_SEC settings*)
		Scope : McASMShSSASSwOntoSegSecScpEnum; (*The scope of the setting*)
	END_STRUCT;
	McASMShSSASAutAttFallbackEnum :
		( (*The fallback strategy if auto attachment fails*)
		mcASMSSSASAAF_SEG_SEC := 0, (*Segment sector - Switch onto segment sector*)
		mcASMSSSASAAF_INT_SEC := 1 (*Internal sector - Remain on internal sector*)
		);
	McASMShSSASAutAttType : STRUCT (*Type mcASMSSSAS_AUT_ATT settings*)
		Fallback : McASMShSSASAutAttFallbackEnum; (*The fallback strategy if auto attachment fails*)
	END_STRUCT;
	McASMShSSASRmnOnIntSecScpEnum :
		( (*The scope of the setting*)
		mcASMSSSASROISS_CON_ONLY := 0, (*Convoy only - The non-trivial convoy remains on the internal sector. The shuttle or trivial convoy switches onto the segment sector*)
		mcASMSSSASROISS_ALL := 1 (*All - The shuttle or convoy remains on the internal sector*)
		);
	McASMShSSASRmnOnIntSecType : STRUCT (*Type mcASMSSSAS_RMN_ON_INT_SEC settings*)
		Scope : McASMShSSASRmnOnIntSecScpEnum; (*The scope of the setting*)
	END_STRUCT;
	McASMShSSASType : STRUCT (*Switch the shuttle or convoy sector if the shuttle or convoy is on an internal sector after stop or error stop*)
		Type : McASMShSSASEnum; (*Switch sector after stop selector setting*)
		SwitchOntoSegmentSector : McASMShSSASSwOntoSegSecType; (*Type mcASMSSSAS_SW_ONTO_SEG_SEC settings*)
		AutoAttach : McASMShSSASAutAttType; (*Type mcASMSSSAS_AUT_ATT settings*)
		RemainOnInternalSector : McASMShSSASRmnOnIntSecType; (*Type mcASMSSSAS_RMN_ON_INT_SEC settings*)
	END_STRUCT;
	McASMShDistResType : STRUCT (*Parameter setting for shuttle distance reserves*)
		CollisionAvoidance : LREAL; (*Safety distance which is added to the distance a shuttle has to keep to obstacles [Measurement units]*)
		ErrorStopAvoidance : LREAL; (*Additional safety distance between shuttles in order to avoid error stops [Measurement units]*)
	END_STRUCT;
	McASMShShSttType : STRUCT (*Parameter settings for the shuttles*)
		ShuttleStereotypeReference : McCfgUnboundedArrayType; (*Name of the shuttle stereotype reference*)
	END_STRUCT;
	McASMShMagnPltCfgShTypEnum :
		( (*Shuttle type 1-1 selector setting*)
		mcASMSMPCST_ST8F1SA100 := 0, (*ST8F1SA100 - 5 magnet poles on both sides of the shuttle*)
		mcASMSMPCST_ST8F1SA102 := 1, (*ST8F1SA102 - 5 magnet poles on one side of the shuttle*)
		mcASMSMPCST_ST8F1SA104 := 2, (*ST8F1SA104 - 5 magnet poles skewed on both sides of the shuttle*)
		mcASMSMPCST_ST8F1SA106 := 3, (*ST8F1SA106 - 5 magnet poles skewed on one side of the shuttle*)
		mcASMSMPCST_ST8F1SA201 := 4, (*ST8F1SA201 - 10 magnet poles on both sides of the shuttle*)
		mcASMSMPCST_ST8F1SA203 := 5, (*ST8F1SA203 - 10 magnet poles on one side of the shuttle*)
		mcASMSMPCST_ST8F1SB308 := 6 (*ST8F1SB308 - 21 magnet poles on one side of the shuttle*)
		);
	McASMShMagnPltCfgShTypType : STRUCT (*Parameters of the magnet plate*)
		Type : McASMShMagnPltCfgShTypEnum; (*Shuttle type 1-1 selector setting*)
	END_STRUCT;
	McASMShMagnPltCfgType : STRUCT (*Parameter settings for the magnet plates*)
		ShuttleType : McCfgUnboundedArrayType; (*Parameters of the magnet plate*)
	END_STRUCT;
	McASMShColAvStratEnum :
		( (*Strategy selector setting*)
		mcASMSCAS_CONST := 0, (*Constant - Constant minimal distance between shuttles*)
		mcASMSCAS_VAR := 1, (*Variable - Variable minimal distance between shuttles*)
		mcASMSCAS_ADV_CONST := 2, (*Advanced constant - Optimized constant minimal distance between shuttles*)
		mcASMSCAS_ADV_VAR := 3 (*Advanced variable - Optimized variable minimal distance between shuttles*)
		);
	McASMShColAvStratType : STRUCT (*Type of active collision avoidance*)
		Type : McASMShColAvStratEnum; (*Strategy selector setting*)
	END_STRUCT;
	McASMShColAvExEnum :
		( (*Exclusion selector setting*)
		mcASMSCAE_NOT_USE := 0, (*Not used - Collision avoidance is active for all physical and virtual shuttles*)
		mcASMSCAE_VIRT_SH := 1, (*Virtual shuttles - Exclude all virtual shuttles from collision avoidance, i.e., do not prevent virtual shuttles from overlapping with any other shuttles*)
		mcASMSCAE_VIRT_TOWARDS_PHS_SH := 2 (*Virtual towards physical shuttles - Exclude virtual shuttles from collision avoidance towards physical shuttles, i.e., do not prevent virtual shuttles from overlapping with any physical shuttles*)
		);
	McASMShColAvExType : STRUCT (*Type of exclusion for collision avoidance*)
		Type : McASMShColAvExEnum; (*Exclusion selector setting*)
	END_STRUCT;
	McASMShColAvMaxMdlDimLenType : STRUCT (*Length of the shuttle model*)
		ExtentToFront : LREAL; (*Extent from the center point of the magnet plate to the front of the shuttle [Measurement units]*)
		ExtentToBack : LREAL; (*Extent from the center point of the magnet plate to the back of the shuttle [Measurement units]*)
	END_STRUCT;
	McASMShColAvMaxMdlDimWidType : STRUCT (*Width of the shuttle model*)
		Width : LREAL; (*Total symmetric width of shuttle and product relative to shuttle center point [Measurement units]*)
	END_STRUCT;
	McASMShColAvMaxMdlDimType : STRUCT (*Maximum model dimensions for calculating the diverters*)
		Length : McASMShColAvMaxMdlDimLenType; (*Length of the shuttle model*)
		Width : McASMShColAvMaxMdlDimWidType; (*Width of the shuttle model*)
	END_STRUCT;
	McASMShColAvType : STRUCT (*Parameter settings for the collision avoidance*)
		Strategy : McASMShColAvStratType; (*Type of active collision avoidance*)
		Exclusion : McASMShColAvExType; (*Type of exclusion for collision avoidance*)
		MaximumModelDimensions : McASMShColAvMaxMdlDimType; (*Maximum model dimensions for calculating the diverters*)
	END_STRUCT;
	McASMShCplgCplgFeatType : STRUCT (*Settings for Cam or GearIn coupling*)
		EliminateShuttleDelay : BOOL; (*Eliminate delay of one cycle when coupling a shuttle to another shuttle*)
	END_STRUCT;
	McASMShCplgType : STRUCT
		CouplingFeature : McASMShCplgCplgFeatType; (*Settings for Cam or GearIn coupling*)
	END_STRUCT;
	McASMShType : STRUCT (*Settings for the shuttles*)
		MaximumCount : UINT; (*Maximum count of shuttles in the assembly*)
		MaximumDelegatedCommandCount : UINT; (*Maximum count of shuttles which start a command triggered by an assembly command within one cycle (0 implies no limit)*)
		DecelerationAtAssemblyCommands : REAL; (*Deceleration used for shuttle stops triggered by assembly commands (0.0 implies using respective axis limits)*)
		ConvoyFunctionality : McASMShConFunEnum; (*Activate for usage of shuttle convoys*)
		SwitchSectorAfterStop : McASMShSSASType; (*Switch the shuttle or convoy sector if the shuttle or convoy is on an internal sector after stop or error stop*)
		DistanceReserves : McASMShDistResType; (*Parameter setting for shuttle distance reserves*)
		ShuttleStereotypes : McASMShShSttType; (*Parameter settings for the shuttles*)
		MagnetPlateConfigurations : McASMShMagnPltCfgType; (*Parameter settings for the magnet plates*)
		CollisionAvoidance : McASMShColAvType; (*Parameter settings for the collision avoidance*)
		Coupling : McASMShCplgType;
	END_STRUCT;
	McASMAsmFeatType : STRUCT (*Features for an assembly*)
		AssemblyFeatureReference : McCfgUnboundedArrayType; (*Name of the assembly feature reference*)
	END_STRUCT;
	McASMVisProcTskCEnum :
		( (*Cyclic task class for command processing*)
		mcASMVPTC_CYC_1 := 1, (*Cyclic #1 - Task class 1*)
		mcASMVPTC_CYC_2 := 2, (*Cyclic #2 - Task class 2*)
		mcASMVPTC_CYC_3 := 3, (*Cyclic #3 - Task class 3*)
		mcASMVPTC_CYC_4 := 4, (*Cyclic #4 - Task class 4*)
		mcASMVPTC_CYC_5 := 5, (*Cyclic #5 - Task class 5*)
		mcASMVPTC_CYC_6 := 6, (*Cyclic #6 - Task class 6*)
		mcASMVPTC_CYC_7 := 7, (*Cyclic #7 - Task class 7*)
		mcASMVPTC_CYC_8 := 8 (*Cyclic #8 - Task class 8*)
		);
	McASMVisType : STRUCT (*Defines for connecting to visualization*)
		MonitoringPV : STRING[250]; (*Name of the process variable of type McAcpTrakAssemblyMonData*)
		ProcessingTaskClass : McASMVisProcTskCEnum; (*Cyclic task class for command processing*)
	END_STRUCT;
	McCfgAsmType : STRUCT (*Main data type corresponding to McCfgTypeEnum mcCFG_ASM*)
		Tracks : McASMTrksType; (*Settings for all tracks that define the assembly*)
		CommonSegmentSettings : McASMCSSType; (*Common settings for all segments in the assembly*)
		Shuttles : McASMShType; (*Settings for the shuttles*)
		AssemblyFeatures : McASMAsmFeatType; (*Features for an assembly*)
		Visualization : McASMVisType; (*Defines for connecting to visualization*)
	END_STRUCT;
	McAFCCplgObjType : STRUCT (*Coupling object*)
		Name : STRING[250]; (*Name of the coupling object*)
		ShuttleCount : UINT; (*Maximum number of simultaneously coupled shuttles*)
		CamAutomatReference : McCfgReferenceType; (*Name of the axis feature reference*)
		CamListReference : McCfgReferenceType; (*Name of the cam list reference*)
	END_STRUCT;
	McCfgAsmFeatCplgType : STRUCT (*Main data type corresponding to McCfgTypeEnum mcCFG_ASM_FEAT_CPLG*)
		CouplingObject : McCfgUnboundedArrayType; (*Coupling object*)
	END_STRUCT;
	McAFSSDShOnSecOrientEnum :
		( (*Orientation of the shuttle*)
		mcAFSSDSOSO_POS := 0, (*Positive - Same orientation as sector*)
		mcAFSSDSOSO_NEG := 1 (*Negative - Opposite orientation to the sector*)
		);
	McAFSSDShOnSecDefEnum :
		( (*Definition selector setting*)
		mcAFSSDSOSD_SNG_SH := 0, (*Single shuttle - Definition of shuttles separately*)
		mcAFSSDSOSD_SET_OF_SH := 1 (*Set of shuttles - Definition of the whole shuttle set*)
		);
	McAFSSDShOnSecDefSngShType : STRUCT (*Type mcAFSSDSOSD_SNG_SH settings*)
		Position : McCfgUnboundedArrayType; (*Position on the sector [Measurement units]*)
	END_STRUCT;
	McAFSSDShOnSecDefSetOfShType : STRUCT (*Type mcAFSSDSOSD_SET_OF_SH settings*)
		StartPosition : LREAL; (*Position of the first shuttle on the sector [Measurement units]*)
		NumberOfShuttles : USINT; (*Number of shuttles on the sector [Measurement units]*)
		DistanceBetweenShuttles : LREAL; (*Distance between consecutive shuttles [Measurement units]*)
	END_STRUCT;
	McAFSSDShOnSecDefType : STRUCT (*Type of shuttle definition*)
		Type : McAFSSDShOnSecDefEnum; (*Definition selector setting*)
		SingleShuttle : McAFSSDShOnSecDefSngShType; (*Type mcAFSSDSOSD_SNG_SH settings*)
		SetOfShuttles : McAFSSDShOnSecDefSetOfShType; (*Type mcAFSSDSOSD_SET_OF_SH settings*)
	END_STRUCT;
	McAFSSDShOnSecType : STRUCT (*Shuttle to be initialized*)
		SectorReference : McCfgReferenceType; (*Name of the referenced sector component*)
		Orientation : McAFSSDShOnSecOrientEnum; (*Orientation of the shuttle*)
		Definition : McAFSSDShOnSecDefType; (*Type of shuttle definition*)
	END_STRUCT;
	McCfgAsmFeatSimShDefType : STRUCT (*Main data type corresponding to McCfgTypeEnum mcCFG_ASM_FEAT_SIM_SH_DEF*)
		ShuttleOnSector : McCfgUnboundedArrayType; (*Shuttle to be initialized*)
	END_STRUCT;
	McAFSTShTrcCfgSecRstEnum :
		( (*Sector restricted*)
		mcAFSTSTCSR_ON := 0, (*On - Sector restricted on*)
		mcAFSTSTCSR_OFF := 1 (*Off - Sector restricted off*)
		);
	McAFSTShTrcCfgType : STRUCT (*Shuttle trace configuration*)
		ShuttleCount : UINT; (*Maximum number of simultaneously traced shuttles*)
		SectorReference : McCfgReferenceType; (*Name of the sector reference*)
		SectorRestricted : McAFSTShTrcCfgSecRstEnum; (*Sector restricted*)
	END_STRUCT;
	McCfgAsmFeatShTraceType : STRUCT (*Main data type corresponding to McCfgTypeEnum mcCFG_ASM_FEAT_SH_TRACE*)
		ShuttleTraceConfiguration : McAFSTShTrcCfgType; (*Shuttle trace configuration*)
	END_STRUCT;
	McAFSAAPrioOrientEnum :
		( (*Orientation of the shuttle*)
		mcAFSAAPO_KEEP_SEG_ORIENT := 0, (*Keep segment orientation - Keep currently assigned orientation*)
		mcAFSAAPO_POS := 1, (*Positive - Same orientation as sector*)
		mcAFSAAPO_NEG := 2 (*Negative - Opposite orientation to the sector*)
		);
	McAFSAAPrioType : STRUCT (*Sector priority definition for the shuttle auto attachment*)
		SectorReference : McCfgReferenceType; (*Name of the referenced sector component*)
		Orientation : McAFSAAPrioOrientEnum; (*Orientation of the shuttle*)
	END_STRUCT;
	McCfgAsmFeatShAutAttType : STRUCT (*Main data type corresponding to McCfgTypeEnum mcCFG_ASM_FEAT_SH_AUT_ATT*)
		Priority : McCfgUnboundedArrayType; (*Sector priority definition for the shuttle auto attachment*)
	END_STRUCT;
	McAFLLScpEnum :
		( (*Scope selector setting*)
		mcAFLLS_ALL_SH := 0, (*All shuttles - Applies to all shuttles, not changeable*)
		mcAFLLS_SNG_SH := 1 (*Single shuttles - Applies only to shuttles which are defined*)
		);
	McAFLLScpSngShType : STRUCT (*Type mcAFLLS_SNG_SH settings*)
		LocalLimitName : STRING[250]; (*Local limit name to use for MC_BR_ShLocalLimitCmd_AcpTrak*)
	END_STRUCT;
	McAFLLScpType : STRUCT (*Defines for which shuttles the local limit applies*)
		Type : McAFLLScpEnum; (*Scope selector setting*)
		SingleShuttles : McAFLLScpSngShType; (*Type mcAFLLS_SNG_SH settings*)
	END_STRUCT;
	McAFLLLocEnum :
		( (*Location selector setting*)
		mcAFLLL_SEC := 0, (*Sector - Location defined by a sector*)
		mcAFLLL_CRV_AREA := 1, (*Curved area - Local limit in all curved areas*)
		mcAFLLL_DUALTRK_AREA := 2 (*Dual-track area - Local limit in all dual-track areas*)
		);
	McAFLLLocSecType : STRUCT (*Type mcAFLLL_SEC settings*)
		SectorReference : McCfgReferenceType; (*Name of the referenced sector component*)
	END_STRUCT;
	McAFLLLocCrvAreaType : STRUCT (*Type mcAFLLL_CRV_AREA settings*)
		CurvatureThreshold : REAL; (*Curvature from which the local limit is valid. Value given in the reciprocal of the radius of curvature. [1/m]*)
	END_STRUCT;
	McAFLLLocType : STRUCT (*Defines the location of the local limit*)
		Type : McAFLLLocEnum; (*Location selector setting*)
		Sector : McAFLLLocSecType; (*Type mcAFLLL_SEC settings*)
		CurvedArea : McAFLLLocCrvAreaType; (*Type mcAFLLL_CRV_AREA settings*)
	END_STRUCT;
	McAFLLMotLimVelEnum :
		( (*Velocity selector setting*)
		mcAFLLMLV_NOT_USE := 0, (*Not used - Velocity limit not used*)
		mcAFLLMLV_BASIC := 1, (*Basic -*)
		mcAFLLMLV_ADV := 2 (*Advanced -*)
		);
	McAFLLMotLimVelBasicType : STRUCT (*Type mcAFLLMLV_BASIC settings*)
		Velocity : REAL; (*Velocity limit in any movement direction [Measurement units/s]*)
	END_STRUCT;
	McAFLLMotLimVelType : STRUCT (*Limit the velocity*)
		Type : McAFLLMotLimVelEnum; (*Velocity selector setting*)
		Basic : McAFLLMotLimVelBasicType; (*Type mcAFLLMLV_BASIC settings*)
	END_STRUCT;
	McAFLLMotLimAccEnum :
		( (*Acceleration selector setting*)
		mcAFLLMLA_NOT_USE := 0, (*Not used - Acceleration limit not used*)
		mcAFLLMLA_BASIC := 1, (*Basic -*)
		mcAFLLMLA_ADV := 2 (*Advanced -*)
		);
	McAFLLMotLimAccBasicType : STRUCT (*Type mcAFLLMLA_BASIC settings*)
		Acceleration : REAL; (*Acceleration limit in any movement direction [Measurement units/s²]*)
	END_STRUCT;
	McAFLLMotLimAccType : STRUCT (*Limit the acceleration*)
		Type : McAFLLMotLimAccEnum; (*Acceleration selector setting*)
		Basic : McAFLLMotLimAccBasicType; (*Type mcAFLLMLA_BASIC settings*)
	END_STRUCT;
	McAFLLMotLimType : STRUCT (*Limits which are effective*)
		Velocity : McAFLLMotLimVelType; (*Limit the velocity*)
		Acceleration : McAFLLMotLimAccType; (*Limit the acceleration*)
	END_STRUCT;
	McAFLLType : STRUCT (*Local limit definition*)
		Scope : McAFLLScpType; (*Defines for which shuttles the local limit applies*)
		Location : McAFLLLocType; (*Defines the location of the local limit*)
		MotionLimits : McAFLLMotLimType; (*Limits which are effective*)
	END_STRUCT;
	McCfgAsmFeatLocLimType : STRUCT (*Main data type corresponding to McCfgTypeEnum mcCFG_ASM_FEAT_LOC_LIM*)
		LocalLimit : McCfgUnboundedArrayType; (*Local limit definition*)
	END_STRUCT;
	McAFESExFromEnum :
		( (*Exclusion from selector setting*)
		mcAFESEF_ASM_PWR_ON := 0 (*Assembly power on - Exclude segments from assembly power on*)
		);
	McAFESExFromAsmPwrOnType : STRUCT (*Type mcAFESEF_ASM_PWR_ON settings*)
		SegmentReference : McCfgUnboundedArrayType; (*Name of the referenced segment component*)
	END_STRUCT;
	McAFESExFromType : STRUCT (*Scope of exclusion*)
		Type : McAFESExFromEnum; (*Exclusion from selector setting*)
		AssemblyPowerOn : McAFESExFromAsmPwrOnType; (*Type mcAFESEF_ASM_PWR_ON settings*)
	END_STRUCT;
	McCfgAsmFeatExSegType : STRUCT (*Main data type corresponding to McCfgTypeEnum mcCFG_ASM_FEAT_EX_SEG*)
		ExclusionFrom : McAFESExFromType; (*Scope of exclusion*)
	END_STRUCT;
	McAFSSRSetLenType : STRUCT (*Length of the shuttle model*)
		ExtentToFront : LREAL; (*Extent from the center point of the magnet plate to the front of the shuttle [Measurement units]*)
		ExtentToBack : LREAL; (*Extent from the center point of the magnet plate to the back of the shuttle [Measurement units]*)
	END_STRUCT;
	McAFSSRSetWidType : STRUCT (*Width of the shuttle model*)
		Width : LREAL; (*Total symmetric width of shuttle and product relative to shuttle center point [Measurement units]*)
	END_STRUCT;
	McAFSSRSetType : STRUCT (*Model dimensions set*)
		Length : McAFSSRSetLenType; (*Length of the shuttle model*)
		Width : McAFSSRSetWidType; (*Width of the shuttle model*)
	END_STRUCT;
	McCfgAsmFeatShShpRegType : STRUCT (*Main data type corresponding to McCfgTypeEnum mcCFG_ASM_FEAT_SH_SHP_REG*)
		Set : McCfgUnboundedArrayType; (*Model dimensions set*)
	END_STRUCT;
	McAFSGSegGrpSegType : STRUCT (*List of segments*)
		SegmentReference : McCfgUnboundedArrayType; (*Name of the referenced segment component*)
	END_STRUCT;
	McAFSGSegGrpType : STRUCT (*Group of segments accessed by assembly functionality*)
		Name : STRING[250]; (*Name of the group*)
		Segments : McAFSGSegGrpSegType; (*List of segments*)
	END_STRUCT;
	McCfgAsmFeatSegGrpType : STRUCT (*Main data type corresponding to McCfgTypeEnum mcCFG_ASM_FEAT_SEG_GRP*)
		SegmentGroup : McCfgUnboundedArrayType; (*Group of segments accessed by assembly functionality*)
	END_STRUCT;
	McSTypEnum :
		( (*Type selector setting*)
		mcST_COMP_SEC := 0, (*Composed sector - Sector defined by segments*)
		mcST_SUB_SEC := 1 (*Sub sector - Sector defined by another sector*)
		);
	McSCSegPosRelToEnum :
		( (*Absolute position from which the position is counted*)
		mcSCSPRT_ST_OF_SEG := 0, (*Start of segment - Positive from start of segment*)
		mcSCSPRT_END_OF_SEG := 1 (*End of segment - Negative from end of segment*)
		);
	McSCSegType : STRUCT (*Begin of the sector*)
		SegmentReference : STRING[250]; (*Name of the referenced segment component*)
		Position : LREAL; (*Position on the segment [Measurement units]*)
		PositionRelativeTo : McSCSegPosRelToEnum; (*Absolute position from which the position is counted*)
	END_STRUCT;
	McSCIntmSegType : STRUCT (*Segments between the start and the end segment*)
		SegmentReference : McCfgUnboundedArrayType; (*Name of the referenced segment component*)
	END_STRUCT;
	McCfgSecCompType : STRUCT (*Main data type corresponding to McCfgTypeEnum mcCFG_SEC_COMP*)
		StartSegment : McSCSegType; (*Begin of the sector*)
		IntermediateSegments : McSCIntmSegType; (*Segments between the start and the end segment*)
		EndSegment : McSCSegType; (*End of the sector*)
	END_STRUCT;
	McSSStPosRelToEnum :
		( (*Absolute position from which the position is counted*)
		mcSSSPRT_ST_OF_SEC := 0, (*Start of sector - Tail of the sector*)
		mcSSSPRT_END_OF_SEC := 1 (*End of sector - Head of the sector*)
		);
	McSSStType : STRUCT (*Begin of the sector*)
		Position : LREAL; (*Position on the sector [Measurement units]*)
		PositionRelativeTo : McSSStPosRelToEnum; (*Absolute position from which the position is counted*)
	END_STRUCT;
	McSSDirEnum :
		( (*Direction of the sub sector*)
		mcSSD_POS := 0, (*Positive - Same direction as sector*)
		mcSSD_NEG := 1 (*Negative - Opposite direction of sector*)
		);
	McCfgSecSubType : STRUCT (*Main data type corresponding to McCfgTypeEnum mcCFG_SEC_SUB*)
		SectorReference : McCfgReferenceType; (*Name of the referenced sector component*)
		Start : McSSStType; (*Begin of the sector*)
		Length : LREAL; (*Length of the sub sector [Measurement units]*)
		Direction : McSSDirEnum; (*Direction of the sub sector*)
	END_STRUCT;
	McSTypType : STRUCT (*Type of the configured sector*)
		Type : McSTypEnum; (*Type selector setting*)
		ComposedSector : McCfgSecCompType; (*Type mcST_COMP_SEC settings*)
		SubSector : McCfgSecSubType; (*Type mcST_SUB_SEC settings*)
	END_STRUCT;
	McCfgSecType : STRUCT (*Main data type corresponding to McCfgTypeEnum mcCFG_SEC*)
		Type : McSTypType; (*Type of the configured sector*)
	END_STRUCT;
	McSSTMeasUnitEnum :
		( (*Measurement unit for the axis*)
		mcSSTMU_M := 5067858 (*Meters*)
		);
	McSSTMoveLimEnum :
		( (*Movement limits selector setting*)
		mcSSTML_INT := 0 (*Internal - Internal definition of limits*)
		);
	McSSTMoveLimIntVelEnum :
		( (*Velocity selector setting*)
		mcSSTMLIV_BASIC := 0 (*Basic -*)
		);
	McSSTMoveLimIntVelBasicType : STRUCT (*Type mcSSTMLIV_BASIC settings*)
		Velocity : REAL; (*Velocity limit in any movement direction [Measurement units/s]*)
	END_STRUCT;
	McSSTMoveLimIntVelType : STRUCT (*Limits for the velocity of the axis*)
		Type : McSSTMoveLimIntVelEnum; (*Velocity selector setting*)
		Basic : McSSTMoveLimIntVelBasicType; (*Type mcSSTMLIV_BASIC settings*)
	END_STRUCT;
	McSSTMoveLimIntAccEnum :
		( (*Acceleration selector setting*)
		mcSSTMLIA_BASIC := 0 (*Basic -*)
		);
	McSSTMoveLimIntAccBasicType : STRUCT (*Type mcSSTMLIA_BASIC settings*)
		Acceleration : REAL; (*Acceleration limit in any movement direction [Measurement units/s²]*)
	END_STRUCT;
	McSSTMoveLimIntAccType : STRUCT (*Limits for the acceleration of the axis*)
		Type : McSSTMoveLimIntAccEnum; (*Acceleration selector setting*)
		Basic : McSSTMoveLimIntAccBasicType; (*Type mcSSTMLIA_BASIC settings*)
	END_STRUCT;
	McSSTMoveLimIntDecEnum :
		( (*Deceleration selector setting*)
		mcSSTMLID_BASIC := 0 (*Basic -*)
		);
	McSSTMoveLimIntDecBasicType : STRUCT (*Type mcSSTMLID_BASIC settings*)
		Deceleration : REAL; (*Deceleration limit in any movement direction [Measurement units/s²]*)
	END_STRUCT;
	McSSTMoveLimIntDecType : STRUCT (*Limits for the deceleration of the axis*)
		Type : McSSTMoveLimIntDecEnum; (*Deceleration selector setting*)
		Basic : McSSTMoveLimIntDecBasicType; (*Type mcSSTMLID_BASIC settings*)
	END_STRUCT;
	McSSTMoveLimIntUpdModEnum :
		( (*Setting for the mode of motion limit (acceleration and deceleration) updates*)
		mcSSTMLIUM_IMMED := 0, (*Immediately - Accept motion limits immediately*)
		mcSSTMLIUM_AVOID_ERR_STOP := 1 (*Avoid error stops - Accept motion limits as soon as error stops can be avoided*)
		);
	McSSTMoveLimIntType : STRUCT (*Type mcSSTML_INT settings*)
		Velocity : McSSTMoveLimIntVelType; (*Limits for the velocity of the axis*)
		Acceleration : McSSTMoveLimIntAccType; (*Limits for the acceleration of the axis*)
		Deceleration : McSSTMoveLimIntDecType; (*Limits for the deceleration of the axis*)
		UpdateMode : McSSTMoveLimIntUpdModEnum; (*Setting for the mode of motion limit (acceleration and deceleration) updates*)
	END_STRUCT;
	McSSTMoveLimType : STRUCT (*Various limit values that will be considered for axis movements*)
		Type : McSSTMoveLimEnum; (*Movement limits selector setting*)
		Internal : McSSTMoveLimIntType; (*Type mcSSTML_INT settings*)
	END_STRUCT;
	McSSTJerkFltrEnum :
		( (*Jerk filter selector setting*)
		mcSSTJF_USE := 0, (*Used - Jerk filter is applied*)
		mcSSTJF_NOT_USE := 1 (*Not used - No jerk filter is applied*)
		);
	McSSTJerkFltrUseType : STRUCT (*Type mcSSTJF_USE settings*)
		JerkTime : REAL; (*Jerk filter time [s]*)
	END_STRUCT;
	McSSTJerkFltrType : STRUCT (*Jerk filter*)
		Type : McSSTJerkFltrEnum; (*Jerk filter selector setting*)
		Used : McSSTJerkFltrUseType; (*Type mcSSTJF_USE settings*)
	END_STRUCT;
	McSSTUsrDatType : STRUCT (*Defines the user data*)
		Size : UINT; (*Size of the user data for one shuttle [Byte]*)
	END_STRUCT;
	McSSTCAIMDEnum :
		( (*Initial model dimensions selector setting*)
		mcSSTCAIMD_USE_MAX_DIM := 0, (*Use maximum dimensions -*)
		mcSSTCAIMD_USE_EXP_VAL := 1 (*Use explicit values -*)
		);
	McSSTCAIMDUseExpValLenType : STRUCT (*Length of the shuttle model*)
		ExtentToFront : LREAL; (*Extent from the center point of the magnet plate to the front of the shuttle [Measurement units]*)
		ExtentToBack : LREAL; (*Extent from the center point of the magnet plate to the back of the shuttle [Measurement units]*)
	END_STRUCT;
	McSSTCAIMDUseExpValWidType : STRUCT (*Width of the shuttle model*)
		Width : LREAL; (*Symmetric width relative to the shuttle center point [Measurement units]*)
	END_STRUCT;
	McSSTCAIMDUseExpValType : STRUCT (*Type mcSSTCAIMD_USE_EXP_VAL settings*)
		Length : McSSTCAIMDUseExpValLenType; (*Length of the shuttle model*)
		Width : McSSTCAIMDUseExpValWidType; (*Width of the shuttle model*)
	END_STRUCT;
	McSSTCAIMDType : STRUCT (*Initial model dimensions for a shuttle*)
		Type : McSSTCAIMDEnum; (*Initial model dimensions selector setting*)
		UseExplicitValues : McSSTCAIMDUseExpValType; (*Type mcSSTCAIMD_USE_EXP_VAL settings*)
	END_STRUCT;
	McSSTColAvType : STRUCT (*Parameter settings for the collision avoidance*)
		InitialModelDimensions : McSSTCAIMDType; (*Initial model dimensions for a shuttle*)
	END_STRUCT;
	McSSTStatTransAutReCtrlEnum :
		( (*Setting of whether a shuttle automatically transits from Disabled to a controlled state if it is controllable*)
		mcSSTSTARC_INACT := 0, (*Inactive - State transitions from Disabled are always controlled by the user*)
		mcSSTSTARC_ACT := 1 (*Active - State transitions from Disabled are done automatically*)
		);
	McSSTStatTransType : STRUCT (*Parameter settings for state transitions*)
		AutomaticReControl : McSSTStatTransAutReCtrlEnum; (*Setting of whether a shuttle automatically transits from Disabled to a controlled state if it is controllable*)
	END_STRUCT;
	McCfgShStereoTypType : STRUCT (*Main data type corresponding to McCfgTypeEnum mcCFG_SH_STEREO_TYP*)
		MeasurementUnit : McSSTMeasUnitEnum; (*Measurement unit for the axis*)
		MeasurementResolution : LREAL; (*Possible resolution of measurement unit that can be achieved [Measurement units]*)
		MovementLimits : McSSTMoveLimType; (*Various limit values that will be considered for axis movements*)
		JerkFilter : McSSTJerkFltrType; (*Jerk filter*)
		UserData : McSSTUsrDatType; (*Defines the user data*)
		CollisionAvoidance : McSSTColAvType; (*Parameter settings for the collision avoidance*)
		StateTransitions : McSSTStatTransType; (*Parameter settings for state transitions*)
	END_STRUCT;
	McSEGSegSecDirEnum :
		( (*Direction of the referenced sector component*)
		mcSEGSSD_POS := 0, (*Positive - Create the segment sector with positive direction*)
		mcSEGSSD_NEG := 1 (*Negative - Create the semgent sector with negative direction*)
		);
	McSEGElongationCompEnum :
		( (*Compensation of segment elongation due to change of temperature*)
		mcSEGEC_USE_ASM_SET := 0, (*Use assembly setting - Use the defined setting from the assembly configuration*)
		mcSEGEC_INACT := 1, (*Inactive - No compensation of segment elongation*)
		mcSEGEC_ACT := 2 (*Active - Compensation of segment elongation*)
		);
	McSEGAsymmetricCurCompEnum :
		( (*Compensation of the asymmetrical load at the middle voltage caused by the current distribution*)
		mcSEGACC_INACT := 0, (*Inactive - No compensation of the asymmetric current load*)
		mcSEGACC_ACT := 1 (*Active - Compensation of the asymmetric current load*)
		);
	McSEGStopReacEnum :
		( (*Stop reaction selector setting*)
		mcSEGSR_USE_ASM_SET := 0, (*Use assembly setting - Use the defined setting from the assembly configuration*)
		mcSEGSR_INDUCT_HALT := 1, (*Induction halt - Shuttle stop by setting current in all segment coils*)
		mcSEGSR_COAST_TO_STANDSTILL := 2 (*Coast to standstill - Shuttle stop by reseting current in all segment coils - stop by friction*)
		);
	McSEGStopReacType : STRUCT (*Reaction in case of certain stop conditions*)
		Type : McSEGStopReacEnum; (*Stop reaction selector setting*)
	END_STRUCT;
	McSEGSpdFltrEnum :
		( (*Speed filter selector setting*)
		mcSEGSF_USE_ASM_SET := 0, (*Use assembly setting - Use the defined setting from the assembly configuration*)
		mcSEGSF_NOT_USE := 1, (*Not used - Speed filter disabled*)
		mcSEGSF_LP_1ST_ORD := 2 (*Lowpass 1st order - Lowpass 1st order speed filter*)
		);
	McSEGSpdFltrLP1stOrdType : STRUCT (*Type mcSEGSF_LP_1ST_ORD settings*)
		FilterTime : REAL; (*Filter time constant [s]*)
	END_STRUCT;
	McSEGSpdFltrType : STRUCT (*Filter for actual speed calculation*)
		Type : McSEGSpdFltrEnum; (*Speed filter selector setting*)
		Lowpass1stOrder : McSEGSpdFltrLP1stOrdType; (*Type mcSEGSF_LP_1ST_ORD settings*)
	END_STRUCT;
	McSEGPosLagMonEnum :
		( (*Position controller lag monitor selector setting*)
		mcSEGPCLM_USE_ASM_SET := 0, (*Use assembly setting - Use the defined setting from the assembly configuration*)
		mcSEGPCLM_INACT := 1, (*Inactive - The position controller lag is not cyclically monitored*)
		mcSEGPCLM_ACT := 2 (*Active - The position controller lag is cyclically monitored*)
		);
	McSEGPosLagMonActType : STRUCT (*Type mcSEGPCLM_ACT settings*)
		WarningLimit : REAL; (*Limit value which leads to a position controller lag warning in case it is exceeded [m]*)
	END_STRUCT;
	McSEGPosLagMonType : STRUCT (*Monitor the position controller lag*)
		Type : McSEGPosLagMonEnum; (*Position controller lag monitor selector setting*)
		Active : McSEGPosLagMonActType; (*Type mcSEGPCLM_ACT settings*)
	END_STRUCT;
	McCfgSegType : STRUCT (*Main data type corresponding to McCfgTypeEnum mcCFG_SEG*)
		SegmentReference : STRING[250]; (*Name of the referenced segment component*)
		SegmentSectorReference : STRING[250]; (*Name of the referenced sector component*)
		SegmentSectorDirection : McSEGSegSecDirEnum; (*Direction of the referenced sector component*)
		ElongationCompensation : McSEGElongationCompEnum; (*Compensation of segment elongation due to change of temperature*)
		AsymmetricCurrentCompensation : McSEGAsymmetricCurCompEnum; (*Compensation of the asymmetrical load at the middle voltage caused by the current distribution*)
		StopReaction : McSEGStopReacType; (*Reaction in case of certain stop conditions*)
		SpeedFilter : McSEGSpdFltrType; (*Filter for actual speed calculation*)
		PositionControllerLagMonitor : McSEGPosLagMonType; (*Monitor the position controller lag*)
	END_STRUCT;
END_TYPE
```

### McDS402AxCfg.typ
```iecst
TYPE
	McDAMEType : STRUCT (*Parameter of hardware elements situated between motor encoder and load which influence the scaling*)
		Gearbox : McCfgGearBoxType; (*Specifies a gearbox by defining the ratio between a gearbox input and output*)
		RotaryToLinearTransformation : McCfgRotToLinTrfType; (*Specifies a transformation factor between the output of the gear and the actual load movement*)
	END_STRUCT;
	McDAESType : STRUCT (*Defines the encoder parameters*)
		IncrementsPerRevolution : DINT; (*Increments per revolution of used encoder*)
	END_STRUCT;
	McDAPAVREnum :
		( (*Position actual value range selector setting*)
		mcDAPAVR_DEF := 0, (*Default - Default range 2^32*)
		mcDAPAVR_SET_MAN := 1 (*Set manually - Limits of 0x6064_PositionActualValue*)
		);
	McDAPAVRSetManType : STRUCT (*Type mcDAPAVR_SET_MAN settings*)
		LowerLimit : DINT; (*Lower limit of 0x6064_PositionActualValue*)
		UpperLimit : DINT; (*Upper limit of 0x6064_PositionActualValue*)
	END_STRUCT;
	McDAPAVRType : STRUCT (*Defines the range of DS402 object 0x6064_Position_actual_value*)
		Type : McDAPAVREnum; (*Position actual value range selector setting*)
		SetManually : McDAPAVRSetManType; (*Type mcDAPAVR_SET_MAN settings*)
	END_STRUCT;
	McDACSVMCycPosModEnum :
		( (*Cyclic position mode on drive when using MC_BR_MoveCyclicPosition*)
		mcDACSVMCPM_INTRPL_POS := 0, (*Interpolated position - 0x6060_ModeOfOperation: 7*)
		mcDACSVMCPM_CYC_SYN_POS := 1 (*Cyclic synchronous position - 0x6060_ModeOfOperation: 8*)
		);
	McDACSVMCycVelModEnum :
		( (*Cyclic velocity mode on drive when using MC_BR_VelocityControl*)
		mcDACSVMCVM_PROF_VEL := 0, (*Profile velocity - 0x6060_ModeOfOperation: 3*)
		mcDACSVMCVM_CYC_SYN_VEL := 1 (*Cyclic synchronous velocity - 0x6060_ModeOfOperation: 9*)
		);
	McDACSVMType : STRUCT (*Modes which are used by the drive to process cyclic set values*)
		CyclicPositionMode : McDACSVMCycPosModEnum; (*Cyclic position mode on drive when using MC_BR_MoveCyclicPosition*)
		CyclicVelocityMode : McDACSVMCycVelModEnum; (*Cyclic velocity mode on drive when using MC_BR_VelocityControl*)
	END_STRUCT;
	McDAAFType : STRUCT (*Features for an axis*)
		FeatureReference : McCfgUnboundedArrayType; (*Name of the axis feature reference*)
	END_STRUCT;
	McCfgDS402AxType : STRUCT (*Main data type corresponding to McCfgTypeEnum mcCFG_DS402_AX*)
		AxisReference : McCfgReferenceType; (*Name of the referenced axis component*)
		MechanicalElements : McDAMEType; (*Parameter of hardware elements situated between motor encoder and load which influence the scaling*)
		EncoderSettings : McDAESType; (*Defines the encoder parameters*)
		PositionActualValueRange : McDAPAVRType; (*Defines the range of DS402 object 0x6064_Position_actual_value*)
		CyclicSetValueModes : McDACSVMType; (*Modes which are used by the drive to process cyclic set values*)
		AxisFeatures : McDAAFType; (*Features for an axis*)
	END_STRUCT;
	McCfgDS402InvAxType : STRUCT (*Main data type corresponding to McCfgTypeEnum mcCFG_DS402_INV_AX*)
		AxisReference : McCfgReferenceType; (*Name of the referenced axis component*)
		MechanicalElements : McDAMEType; (*Parameter of hardware elements situated between motor encoder and load which influence the scaling*)
	END_STRUCT;
	McCfgDS402AxRefType : STRUCT (*Main data type corresponding to McCfgTypeEnum mcCFG_DS402_AX_REF*)
		AxisReference : McCfgReferenceType; (*Name of the referenced axis component*)
	END_STRUCT;
	McCfgDS402AxMechElmType : STRUCT (*Main data type corresponding to McCfgTypeEnum mcCFG_DS402_AX_MECH_ELM*)
		MechanicalElements : McDAMEType; (*Parameter of hardware elements situated between motor encoder and load which influence the scaling*)
	END_STRUCT;
	McCfgDS402AxEncSetType : STRUCT (*Main data type corresponding to McCfgTypeEnum mcCFG_DS402_AX_ENC_SET*)
		EncoderSettings : McDAESType; (*Defines the encoder parameters*)
	END_STRUCT;
	McCfgDS402AxPosActValRngType : STRUCT (*Main data type corresponding to McCfgTypeEnum mcCFG_DS402_AX_POS_ACT_VAL_RNG*)
		PositionActualValueRange : McDAPAVRType; (*Defines the range of DS402 object 0x6064_Position_actual_value*)
	END_STRUCT;
	McCfgDS402AxCycSetValModType : STRUCT (*Main data type corresponding to McCfgTypeEnum mcCFG_DS402_AX_CYC_SET_VAL_MOD*)
		CyclicSetValueModes : McDACSVMType; (*Modes which are used by the drive to process cyclic set values*)
	END_STRUCT;
	McCfgDS402AxFeatType : STRUCT (*Main data type corresponding to McCfgTypeEnum mcCFG_DS402_AX_FEAT*)
		AxisFeatures : McDAAFType; (*Features for an axis*)
	END_STRUCT;
	McCfgAcpInvAxType : STRUCT (*Main data type corresponding to McCfgTypeEnum mcCFG_ACP_INV_AX*)
		AxisReference : McCfgReferenceType; (*Name of the referenced axis component*)
		MechanicalElements : McDAMEType; (*Parameter of hardware elements situated between motor encoder and load which influence the scaling*)
	END_STRUCT;
	McCfgAcpInvAxRefType : STRUCT (*Main data type corresponding to McCfgTypeEnum mcCFG_ACP_INV_AX_REF*)
		AxisReference : McCfgReferenceType; (*Name of the referenced axis component*)
	END_STRUCT;
	McCfgAcpInvAxMechElmType : STRUCT (*Main data type corresponding to McCfgTypeEnum mcCFG_ACP_INV_AX_MECH_ELM*)
		MechanicalElements : McDAMEType; (*Parameter of hardware elements situated between motor encoder and load which influence the scaling*)
	END_STRUCT;
END_TYPE
```

### Program Logical/Program

#### Main.st
```iecst
PROGRAM _INIT

MpDelta4Axis_0.Enable := TRUE;

MpDelta4Axis_0.Override := 100.0;
DeltaParameters.ProgramName := 'Robotic.st';    //File stored on FileDevice

END_PROGRAM

PROGRAM _CYCLIC
//gAxisQ1;
//gAxisQ2;
//gAxisQ3;
//gAxisQ4;

MpDelta4Axis_0.MpLink := ADR(g4AxDeltaA);
MpDelta4Axis_0.Parameters := ADR(DeltaParameters);
MpDelta4Axis_0();

END_PROGRAM
```

### Program Logical/VisionControl

#### Main.st
```iecst
PROGRAM _INIT
	(* Insert code here *)

END_PROGRAM

PROGRAM _CYCLIC
	(* Insert code here *)

END_PROGRAM

PROGRAM _EXIT
	(* Insert code here *)

END_PROGRAM
```

Listed in the project but not available here: Logical/Global.typ, Logical/Camera/Vision/Types.typ, Logical/Camera/Kamera/Types.typ
